(* CODESYS project SGS V4.project
   Description: Diese Software wurde während der Bachelorarbeit für das Strom-Generatorsystem entwickelt.
   Company: Zoyce GmbH
   Version: 4.0
   Title: Strom-Generatorsystem
   Author: Julian Städeli

Project tree, tasks and I/O mapping:
  PLC_AC500_V3 : PM5052-R-ETH, ABB AG, order no. 1SAP124100R0x72, version 3.7.0.0
    application Application
      libraries: Util, * (System); CAA Mathematics, * (CAA Technical Workgroup); VisuElemBase, 4.4.0.0 (System); OnboardIO, * (ABB); VisuDialogs, * (System); SysFile, * (System); SysTimeRtc, * (System); CAA File, * (CAA Technical Workgroup); CAA DTUtil Extern, * (CAA Technical Workgroup); CAA Types Extern, * (CAA Technical Workgroup); SysTime, 3.5.17.0 (System); CAA Memory, * (CAA Technical Workgroup); SysTypes Interfaces, * (System); MQTT Client SL, 1.9.0.0 (CODESYS)
      task Task (cyclic, interval 10 ms, priority 14, watchdog t#20ms x 1) calls Ueberwachung, SunSpec_client, Inverter, Berechnungen, Systemzustand, MQTTDataLogger
      task VISU_TASK (cyclic, interval 100 ms, priority 16) calls VisuElems.Visu_Prg
      CheckConfigurationObject
      program PLC_PRG [ST]
      Diagnosis/
        text list Diag_IO_Bus
        text list Diag_V3_PLC
      trace Trace_Drehzahl (task Task): GV.sys_Drehzahl, GV.sys_Drehzahl_Sensor, GV.sys_Drehzahl_Estimator, GV.sys_Drehzahl_Rechner
      trace Trace_Leistung (task Task): GV.r_LeistungAC, GV.r_LeistungDC
      Symbols
    OnBoard_IO : 12DI/6DO-R/2DC, ABB AG, version 3.7.0.0
        unmapped channels: Fast inputs DI0-DI3, %IB1 Fast inputs DI4-DI7, Standard inputs DI8-DI11, Digital configurable inputs DC12-DC13, Relay outputs NO0-NO3, Relay outputs NO4-NO5 - Digital configurable outputs DC12-DC13
    IO_Bus : I/O-Bus, ABB AG, version 3.7.0.0
    Interfaces : Schnittstellen, ABB AG, version 3.7.0.0
      OptionSlot_1
      OptionSlot_2
      OptionSlot_3
      Ethernet : Ethernet, ABB AG, version 3.7.0.0
        ETH1 : IP-Einstellungen, ABB AG, version 3.7.0.0
          NetConfig : NetzKonfig, ABB AG, version 3.7.0.0
          Web_Server : Webserver, ABB AG, version 3.7.0.0
        Protocols : Client-Protokolle, ABB AG, version 3.7.0.0
          Modbus_TCP_IP_Client : Modbus TCP/IP Client, ABB AG, version 3.7.0.0
    OnBoard_RTC : OnBoardRTC, ABB AG, version 3.7.0.0
  libraries: VisuSymbols, 4.4.0.0 (System); VisuDialogs, * (System); CmpBitmapPool, 3.5.17.0 (System); SysFile, 3.5.17.0 (System); SysFile, 1.0.3.1 (ABB); CAA DTUtil Extern, 3.5.17.0 (CAA Technical Workgroup); SysTypes, 3.1.2.0 (System); SysTypes Interfaces, * (System); SysTimeRtc, 3.5.17.0 (System); CAA File, 3.5.19.0 (CAA Technical Workgroup); MQTT Client SL, 1.9.0.0 (CODESYS)
  global variables GV
  program Schaltlogik [FBD]
  program Ueberwachung [FBD]
  text list GlobalTextList
  program SunSpec_client [FBD]
  data type SunSpec_Model_Inverter1
  SunSpec_Translator/
    function block SunSpec_Write [FBD]
    function block SunSpec_Model_Inverter [ST]
    function block SunSpec_Model_Settings [ST]
    function block SunSpec_Model_Status [ST]
    function block SunSpec_Model_Controls [ST]
    function block SunSpec_Model_MPPT [ST]
    function block SunSpec_Model_Meter [ST]
  program Inverter [ST]
  program Berechnungen [ST]
  image pool ImagePool
  Visualisierung/
    visualisation Uebersicht
    visualisation Elektrotechnik
    visualisation System
    visualisation Parameter
    visualisation Show
    visualisation Logging
    visualisation Info
  5ce3da45-db07-42e7-a21c-a00fff4ed8f6|C:\Users\julia\OneDrive - FHNW\Pro5E\Bilder\Uebersicht Visu.png
  program Systemzustand [ST]
  function block FB_DataLogger [ST]
  5ce3da45-db07-42e7-a21c-a00fff4ed8f6|C:\Users\julia\Downloads\Visu_Show.png
  function WSTRING_TO_BYTEARRAY_UTF8 [ST]
  function block FB_MQTT_Logger [ST]
  function WSTRING_Concat [ST]
  program MQTTDataLogger [ST]
*)

// SunSpec_Model_Inverter1
TYPE SunSpec_Model_Inverter1 :
STRUCT
	ID	:INT;
	Length	:INT;
	AC_Current	:INT;
	Phase_A_Current	:REAL;
	Phase_B_Current	:REAL;
	Phase_C_Current	:REAL;
	
	Phase_Voltage_AB	:REAL;
	Phase_Voltage_BC	:REAL;
	Phase_Voltage_CA	:REAL;
	Phase_Voltage_AN	:REAL;
	Phase_Voltage_BN	:REAL;
	Phase_Voltage_CN	:REAL;
	
	AC_Power	:REAL;
	AC_Frequency	:REAL;
	
	AC_Apparent_Power	:REAL;
	AC_Reactive_Power	:REAL;
	AC_PowerFactor		:REAL;
	AC_Energy			:REAL;
	
	DC_Power	:REAL;
	Temperature :REAL;

	
	
	
	
	
	
	
	
	
	
	
	
END_STRUCT
END_TYPE

// GV
{attribute 'qualified_only'}
(*
Diese Software rurde für die Bachelorarbeit "Stromerzeugungssystem für ein Kleinwasserkraftwerk" 
an der Fachhochschule Nordwestschweiz (FHNW) entwickelt.

Diplomand:		Julian Städeli
				julian.staedeli@students.fhnw.ch	|	julian@staedelis.com
Dozent:			Georg Traxler-Samek
				georg.traxlersamek@fhnw.ch
				
*)

VAR_GLOBAL
	
// Inputs
I_Notaus 			AT %IX0.0		:BOOL;		// I0 Not-Aus Kontakt
I_Steuerspannung 	AT %IX0.1		:BOOL;		// I1 Ausgang Relais Steuerspannung
I_Einschalten 		AT %IX0.2		:BOOL;		// I2 Kontakt Einschalttaster
I_Ausschalten 		AT %IX0.3		:BOOL;		// I3 Kontakt Ausschalttaster
I_Sensor_Drehzahl 	AT %IX1.0		:BOOL;		// I4 Kontakt Sensor, Induktiver Näherungsschalter
I_Hauptschuetz 		AT %IX1.1		:BOOL;		// I5 Hilfskontakt Hauptschütz
I_Ladeschuetz 		AT %IX1.2		:BOOL;		// I6 Hilfskontakt Ladeschütz
I_Motorschutz 		AT %IX1.3		:BOOL;		// I7 Hilfskontakt Motorschutzschalter
I_Temperatur 		AT %IX2.0		:BOOL;		// I8 Thermokontakt im Generator

I_Counter							:UDINT;		// Fast Counter für Sensor

 //AT %IX3.0

// Outputs
O_Steuerspannung	AT %QX0.1		:BOOL;		// NO1 Relais Steuerspannung
O_Infolampe			AT %QX0.2		:BOOL;		// NO2 Infolampe auf Bedienfeld 
O_Hauptschuetz 		AT %QX0.3		:BOOL;		// NO3 Hauptschütz
O_Ladeschuetz		AT %QX1.0		:BOOL;		// NO4 Ladeschütz


// Störungen
stoerung_Notaus				:BOOL;
stoerung_Steuerspannung		:BOOL;
stoerung_Hauptschuetz		:BOOL;
stoerung_Ladeschuetz		:BOOL;
stoerung_Motorschutz		:BOOL;
stoerung_Inverter			:BOOL;
stoerung_Temperatur			:BOOL;

stoerung_Drehzahl			:BOOL;
sammelstoerung				:BOOL;
stoerung_quittieren			:BOOL;

stoerung_Modbus_Lesen		:BOOL;
stoerung_Modbus_Schreiben	:BOOL;
stoerung_MQTT				:BOOL;


// Zustände System
sys_Einschalten				:BOOL;				// Einschaltbefehl
sys_Ausschalten				:BOOL;				// Auschaltbefehl

sys_aus						:BOOL :=TRUE;		// System ist aus: Inverter Heruntergefahren, Schütze offen, Geni im Leerlauf
sys_start					:BOOL;				// Einschaltprozess mit Ladeschaltung und Hochfahren des Inverters
sys_bereit					:BOOL;				// System bereit zum Produzieren
sys_betrieb					:BOOL;				// System läuft 
sys_herunterfahren			:BOOL;				// System wird heruntergefahren

sys_MPPT_aktiv				:BOOL;		// System soll über MPPT arbeiten / befindet sich im Automatikbetrieb
sys_MPP_erreicht			:BOOL;				// Gibt an, ob sich der Tracker am MPP befindet.
sys_LeistungBegrenzung 		:UINT;				// Die eingestellte Leistung, die dem Inverter als Begrenzung übergeben wird (Wert 100 = 10% von 3000W)
			
sys_Drehzahl_Sensor			:REAL;				// Berechnete Drehzahl über Sensor
sys_Drehzahl_Estimator		:REAL;				// Berechnete Drehzahl über der gemessenen Spannung
sys_Drehzahl_Rechner		:REAL;				// Berechnete Drehzahl über Ersatzschaltbild
sys_Drehzahl				:REAL; 				// Systemdrehzahl, die von dem Programm genutzt wird (über Parameter einstellbar)
sys_Drehzahl_Wasserrad		:REAL;				// Berechnete Drehzahl des Wasserrads

// Inverter

// Zustände Inverter
r_StateCode					:STRING; 			// Aus / Standby / Startet / Arbeitet
r_Status					:STRING;
r_Begrenzung				:STRING; 			// Ein / Aus

inv_herunterfahren			:BOOL;				// Inverter soll ausgeschaltet werden
inv_ein						:BOOL;				// Ist eingeschaltet
inv_bereit					:BOOL;				// Ist hochgefahren 
inv_betrieb					:BOOL;				// produziert
inv_leerlauf				:BOOL;				// Ist eingekoppelt aber keine produktion
inv_standby					:BOOL;
inv_fehler					:BOOL;
inv_MaxLeistungEingestellt 	:REAL;				// Eingestellte Leistungsbegrenzung



// Visu
v_LeistungBegrenzung		:UINT;				// Eingestellte Leistung über Visu [W]
v_LeistungBegrenzung_ein	:BOOL;				// Begrenzung mit Visu forcieren

v_Einschalten				:BOOL;				// Einschaltbefehl über Visu
v_Ausschalten				:BOOL;				// Ausschaltbefehl über Visu
v_Notaus					:BOOL;				// Notaus üner Visu
v_Geni_lauft				:BOOL;				// Es wird eine Drehzahl gemessen


	// Modbus 
inv_IP						:STRING;			// IP-Adresse des Inverter, z. B. '192.168.0.51'


	// Daten Modbus (readings)
	//Inverter
r_StromPhaseA				:REAL;		// [A]
r_StromPhaseB				:REAL;		// [A]
r_StromPhaseC				:REAL;		// [A]
r_StrangspannungA			:REAL;		// [V]
r_StrangspannungB			:REAL;		// [V]
r_StrangspannungC			:REAL;		// [V]
r_SpannungPCC				:REAL;		// [V]

r_Frequenz					:REAL;		// [Hz]
r_LeistungAC				:REAL;		// [W]
r_PF						:REAL;
r_Energie					:REAL;		// [Wh]

r_StromDC					:REAL;		// [A]
r_SpannungDC				:REAL;		// [V]
r_LeistungDC				:REAL;		// [W]
r_EnergieDC					:REAL;		// [Wh]		

r_Temperatur				:REAL;		// [°C]

r_MaxLeistung				:REAL;		// [W]

 // Smartmeter
 r_sm_Leistung				:REAL;


	// Befehle Modbus (write)
w_Einschalten				:UINT :=1;	// Inverter soll Einschalten
w_LeistungBegrenzung		:UINT;		// Entweder über Visu oder MPPT vorgegebene Leistungsbegrenzung [%]
w_RampTime	 				:UINT;		// Zeitintervall von einem punkt zum nächsten (funktioniert nicht) [s]
w_Standby					:UINT;		// Inverter soll Ausschalten

	// Überprüfung der Eingestellten Werte
r_Einschalten				:INT;
r_LeistungBegrenzung		:REAL;		
r_RampTime					:REAL;	
r_Standby					:STRING;	




// Parameter
p_Inverter_IP		:STRING :='192.168.178.45';		// IP-Adresse des Inverter, z. B. '192.168.0.51'

p_Drehzahl_soll		:INT :=360;						// Sollwert für Drehzahlregulierung [rpm]					
p_Drehzahl_Toleranz	:INT :=5;						// Angenommene Ungenauigkeit [rpm]
p_Drehzahl_max		:INT :=690;						// Maximal erlaubte Drehzahl [rpm]
p_Drehzahl_min		:INT :=200;						// Minimal benötigte Drehzahl [rpm]
p_Sensor_Impulse	:INT := 4;						// Anzahl Impulse pro rpm die der Sensor liefert [1/rpm]
p_Sensor_Intervall	:TIME := T#1S;					// Wie lange die Impulse vor der Berechnung gemacht werden

p_Leistung_Init		:UINT := 200;					// Mit welcher Leistung gestartet wird [100.00% = 10000]
p_Leistung_Toleranz	:REAL :=30;						// Erlaubte Abweichung, damit es als erreicht gilt [W]
p_Leistung_Anpassung :REAL := 10;					// Leistungsanpassungsschritt [00.10%= 10]

p_MPPT_Intervall	:TIME := T#3S;					// Wie lange gewartet wird, bis MPP einen nächsten Schritt macht [s]
p_MPPT_Timeout		:TIME :=T#3S;					// Wie lange, bis die Leistung als  nicht erreicht betrachtet wird [s]

p_Automatik			:BOOL := TRUE; 					// System fährt selbständig hoch und runter

p_Herunterfahren_Intervall	:TIME := T#1S;			// Wie langae zwischen den Schritten gewartet wird [s]

timenow			:DATE_AND_TIME;


// Show
v_speicher_start	:BOOL := TRUE;
v_Kaffeemaschine :REAL;
v_speicher :REAL :=0;

log_time :ARRAY[1..2000] OF REAL;
log_DrehzahlSoll :ARRAY[1..2000] OF REAL;
log_DrehzahlIst :ARRAY[1..2000] OF REAL;
log_Leistung :ARRAY[1..2000] OF REAL;

END_VAR

// Ueberwachung
PROGRAM Ueberwachung
VAR
	zeit_bis_stoerung :TIME :=t#1s;
	RS_Notaus: RS;
	TON_stoerung_Steuerspannung: TON;
	RS_stoerung_Steuerspannung: SR;
	TON_stoerung_Hauptschuetz: TON;
	RS_stoerung_Hauptschuetz: RS;
	TON_stoerung_Ladeschuetz: TON;
	RS_stoerung_Ladeschuetz: RS;
	RS_Motorschutz: RS;
	RS_Sammelstoerung: RS;
	TON_quittieren: TON;
	RS_Drehzahl: RS;
	TON_Drehzahl: TON;
	RS_Temperatur: RS;
	SR_Notaus: SR;
	SR_stoerung_Steuerspannung: SR;
	SR_stoerung_Hauptschuetz: SR;
	SR_stoerung_Ladeschuetz: SR;
	SR_Motorschutz: SR;
	SR_Temperatur: SR;
	SR_Drehzahl: SR;
	SR_Sammelstoerung: SR;
END_VAR

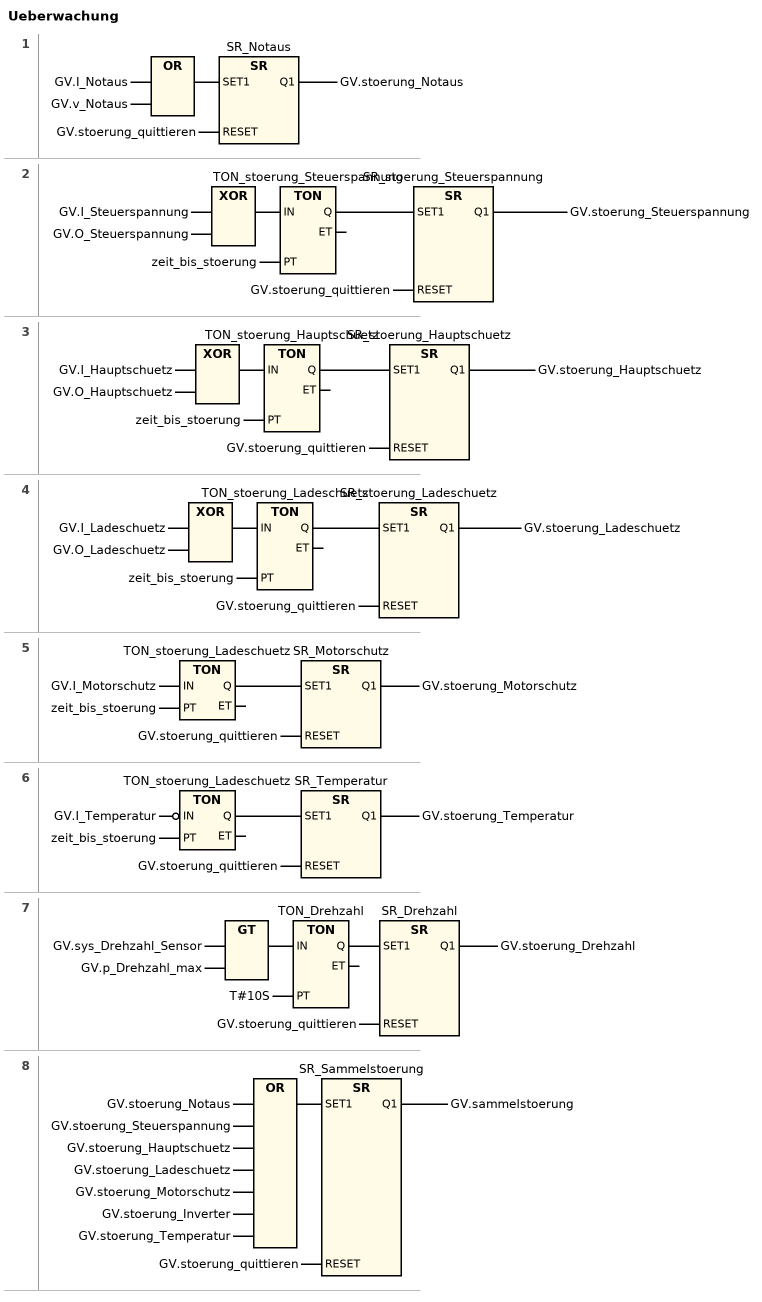
// NETWORK 1
SR_Notaus(SET1 := GV.I_Notaus OR GV.v_Notaus, RESET := GV.stoerung_quittieren); // SR
GV.stoerung_Notaus := SR_Notaus.Q1;

// NETWORK 2
TON_stoerung_Steuerspannung(IN := GV.I_Steuerspannung XOR GV.O_Steuerspannung, PT := zeit_bis_stoerung); // TON
SR_stoerung_Steuerspannung(SET1 := TON_stoerung_Steuerspannung.Q, RESET := GV.stoerung_quittieren); // SR
GV.stoerung_Steuerspannung := SR_stoerung_Steuerspannung.Q1;

// NETWORK 3
TON_stoerung_Hauptschuetz(IN := GV.I_Hauptschuetz XOR GV.O_Hauptschuetz, PT := zeit_bis_stoerung); // TON
SR_stoerung_Hauptschuetz(SET1 := TON_stoerung_Hauptschuetz.Q, RESET := GV.stoerung_quittieren); // SR
GV.stoerung_Hauptschuetz := SR_stoerung_Hauptschuetz.Q1;

// NETWORK 4
TON_stoerung_Ladeschuetz(IN := GV.I_Ladeschuetz XOR GV.O_Ladeschuetz, PT := zeit_bis_stoerung); // TON
SR_stoerung_Ladeschuetz(SET1 := TON_stoerung_Ladeschuetz.Q, RESET := GV.stoerung_quittieren); // SR
GV.stoerung_Ladeschuetz := SR_stoerung_Ladeschuetz.Q1;

// NETWORK 5
TON_stoerung_Ladeschuetz(IN := GV.I_Motorschutz, PT := zeit_bis_stoerung); // TON
SR_Motorschutz(SET1 := TON_stoerung_Ladeschuetz.Q, RESET := GV.stoerung_quittieren); // SR
GV.stoerung_Motorschutz := SR_Motorschutz.Q1;

// NETWORK 6
TON_stoerung_Ladeschuetz(IN := NOT GV.I_Temperatur, PT := zeit_bis_stoerung); // TON
SR_Temperatur(SET1 := TON_stoerung_Ladeschuetz.Q, RESET := GV.stoerung_quittieren); // SR
GV.stoerung_Temperatur := SR_Temperatur.Q1;

// NETWORK 7
TON_Drehzahl(IN := GV.sys_Drehzahl_Sensor > GV.p_Drehzahl_max, PT := T#10S); // TON
SR_Drehzahl(SET1 := TON_Drehzahl.Q, RESET := GV.stoerung_quittieren); // SR
GV.stoerung_Drehzahl := SR_Drehzahl.Q1;

// NETWORK 8
SR_Sammelstoerung(SET1 := GV.stoerung_Notaus OR GV.stoerung_Steuerspannung OR GV.stoerung_Hauptschuetz OR GV.stoerung_Ladeschuetz OR GV.stoerung_Motorschutz OR GV.stoerung_Inverter OR GV.stoerung_Temperatur, RESET := GV.stoerung_quittieren); // SR
GV.sammelstoerung := SR_Sammelstoerung.Q1;

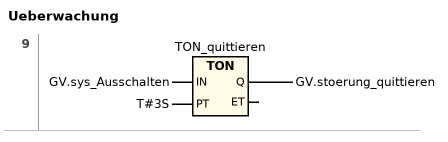
// NETWORK 9
TON_quittieren(IN := GV.sys_Ausschalten, PT := T#3S); // TON
GV.stoerung_quittieren := TON_quittieren.Q;

END_PROGRAM

// SunSpec_client
PROGRAM SunSpec_client
VAR
	inverterIP :STRING := GV.p_Inverter_IP;
// SunSpec Adressen für das Auslesen
	// SunSpec_Adr_Model_Common :WORD := 40003;
	SunSpec_Adr_Model_Inverter :WORD := 40070;
	// SunSpec_Adr_Model_Nameplate :WORD := 40122;
	SunSpec_Adr_Model_Settings :WORD := 40150;
	SunSpec_Adr_Model_Status	:WORD := 40182;
	SunSpec_Adr_Model_Controls :WORD := 40228;
	SunSpec_Adr_Model_MPPT		:WORD := 40254;
	SunSpec_Adr_Model_AC_Meter	:WORD := 40070;
// Buffer für Lesedaten
	inverterData_Inverter AT %MW10 : ARRAY[1..50] OF INT;
	inverterData_Settings AT %MW60 :ARRAY [1..30] OF INT;
	inverterData_Status AT %MW90 :ARRAY [1..50] OF INT;
	inverterData_Controls AT %MW140:ARRAY [1..30] OF INT;
	inverterData_MPPT AT %MW170 :ARRAY [1..30] OF INT;	
	meterData_Main AT %MW200 :ARRAY [1..75] OF INT;

	
// SunSpec Adressen für das Schreiben	
	SunSpec_Adr_Connection	:WORD := 40232;
	SunSpec_Adr_MaxPower	:WORD := 40233;
	SunSpec_Adr_RampTime		:WORD := 40236;
	SunSpec_Adr_Throttle	:WORD := 40237;
// Buffer für Schreibdaten
	inverterCommand_Connection 	AT %MW1		:UINT := GV.w_Einschalten;
	inverterCommand_maxPower 	AT %MW2		:UINT := GV.w_LeistungBegrenzung;
	inverterCommand_RampTime 	AT %MW3		:UINT := GV.w_RampTime;
	inverterCommand_Throttle 	AT %MW4		:UINT :=1;

	clk_Pulse :TIME := T#900MS;
	
	clock: BLINK;
	SunSpec_Inverter: modTcpMast2;
	SunSpec_Settings: ModTcpMast2;
	SunSpec_Controls: modTcpMast2;
	SunSpec_MPPT: modTcpMast2;
	SunSpec_Status: modTcpMast2;
	SunSpec_Write: modTcpMast2;
	SunSpec_Model_Inverter_0: SunSpec_Model_Inverter;
	SunSpec_Model_Settings_0: SunSpec_Model_Settings;
	SunSpec_Model_Status_0: SunSpec_Model_Status;
	SunSpec_Model_Controls_0: SunSpec_Model_Controls;
	SunSpec_Model_MPPT_0: SunSpec_Model_MPPT;
	R_TRIG_0: R_TRIG;
	SunSpec_Write1: modTcpMast2;
	SunSpec_Write2: modTcpMast2;
	SunSpec_Write_0: SunSpec_Write;
	SunSpec_Meter_main: modTcpMast2;
	SunSpec_Meter_Generator: modTcpMast2;
	SunSpec_Model_Meter_main: SunSpec_Model_Meter;
	SunSpec_Model_Meter_generator: SunSpec_Model_Meter;
END_VAR

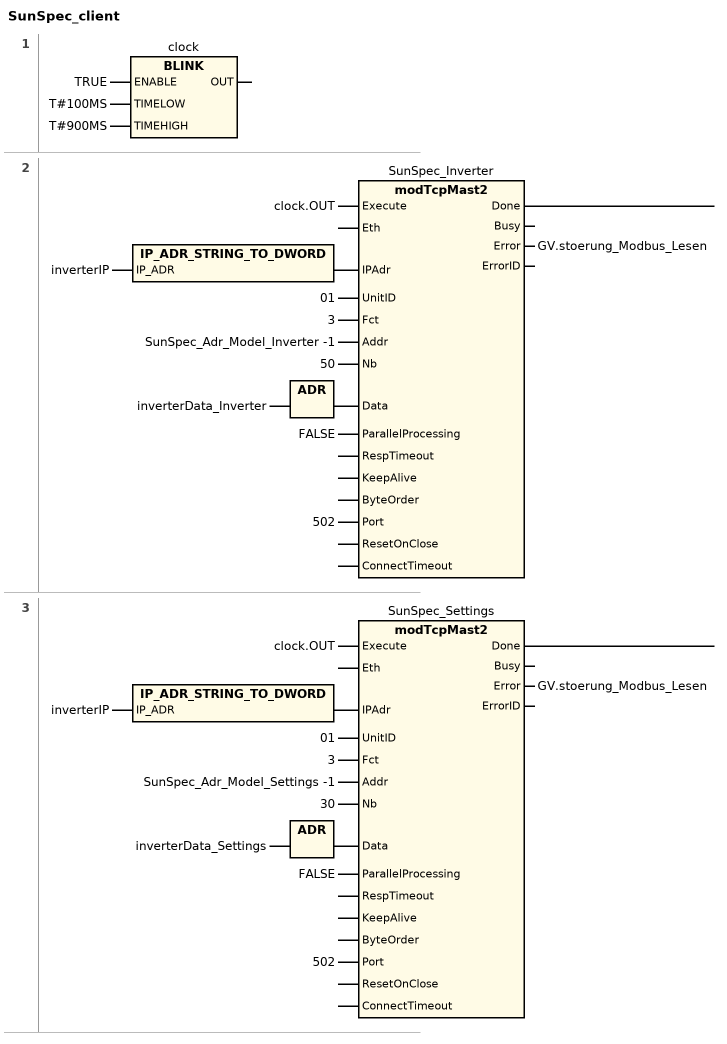
// NETWORK 1
clock(ENABLE := TRUE, TIMELOW := T#100MS, TIMEHIGH := T#900MS); // BLINK

// NETWORK 2
SunSpec_Inverter(
    Execute := clock.OUT,
    IPAdr := IP_ADR_STRING_TO_DWORD(IP_ADR := inverterIP),
    UnitID := 01,
    Fct := 3,
    Addr := SunSpec_Adr_Model_Inverter -1,
    Nb := 50,
    Data := ADR(inverterData_Inverter),
    ParallelProcessing := FALSE,
    Port := 502,
    Error => GV.stoerung_Modbus_Lesen); // modTcpMast2

// NETWORK 3
SunSpec_Settings(
    Execute := clock.OUT,
    IPAdr := IP_ADR_STRING_TO_DWORD(IP_ADR := inverterIP),
    UnitID := 01,
    Fct := 3,
    Addr := SunSpec_Adr_Model_Settings -1,
    Nb := 30,
    Data := ADR(inverterData_Settings),
    ParallelProcessing := FALSE,
    Port := 502,
    Error => GV.stoerung_Modbus_Lesen); // modTcpMast2

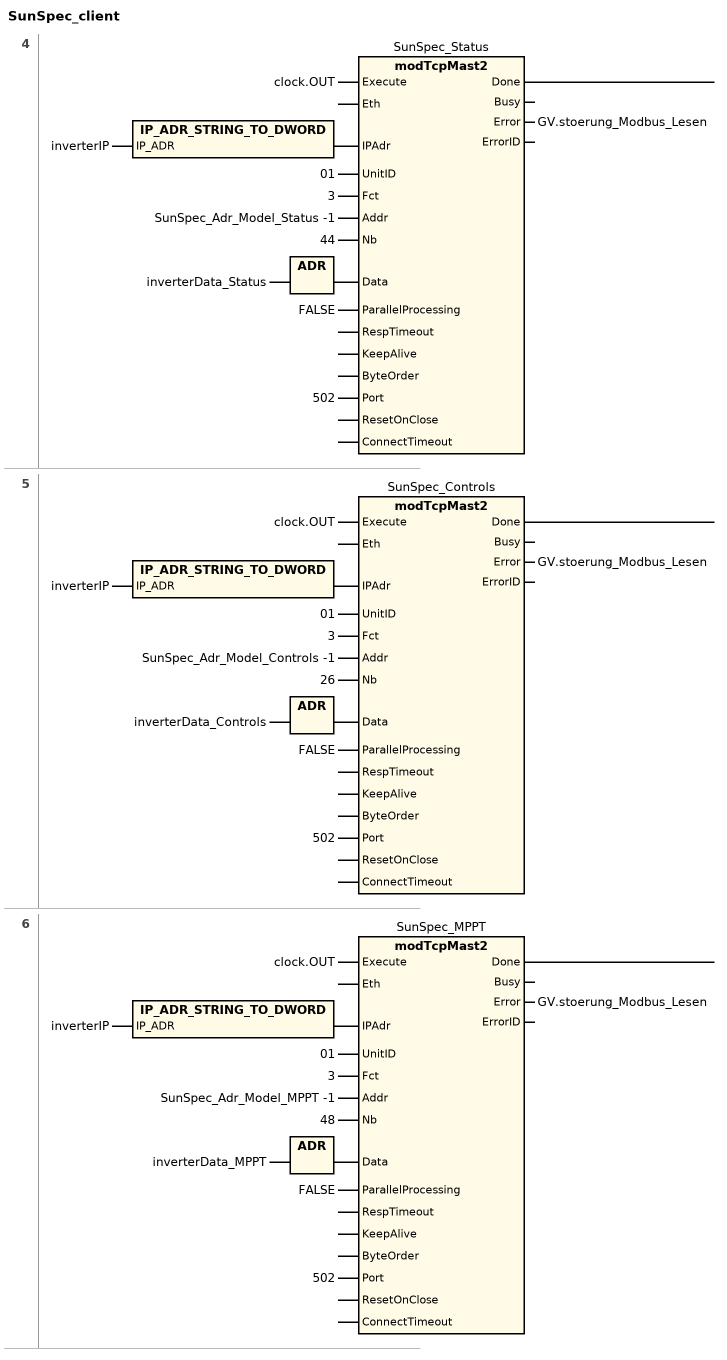
// NETWORK 4
SunSpec_Status(
    Execute := clock.OUT,
    IPAdr := IP_ADR_STRING_TO_DWORD(IP_ADR := inverterIP),
    UnitID := 01,
    Fct := 3,
    Addr := SunSpec_Adr_Model_Status -1,
    Nb := 44,
    Data := ADR(inverterData_Status),
    ParallelProcessing := FALSE,
    Port := 502,
    Error => GV.stoerung_Modbus_Lesen); // modTcpMast2

// NETWORK 5
SunSpec_Controls(
    Execute := clock.OUT,
    IPAdr := IP_ADR_STRING_TO_DWORD(IP_ADR := inverterIP),
    UnitID := 01,
    Fct := 3,
    Addr := SunSpec_Adr_Model_Controls -1,
    Nb := 26,
    Data := ADR(inverterData_Controls),
    ParallelProcessing := FALSE,
    Port := 502,
    Error => GV.stoerung_Modbus_Lesen); // modTcpMast2

// NETWORK 6
SunSpec_MPPT(
    Execute := clock.OUT,
    IPAdr := IP_ADR_STRING_TO_DWORD(IP_ADR := inverterIP),
    UnitID := 01,
    Fct := 3,
    Addr := SunSpec_Adr_Model_MPPT -1,
    Nb := 48,
    Data := ADR(inverterData_MPPT),
    ParallelProcessing := FALSE,
    Port := 502,
    Error => GV.stoerung_Modbus_Lesen); // modTcpMast2

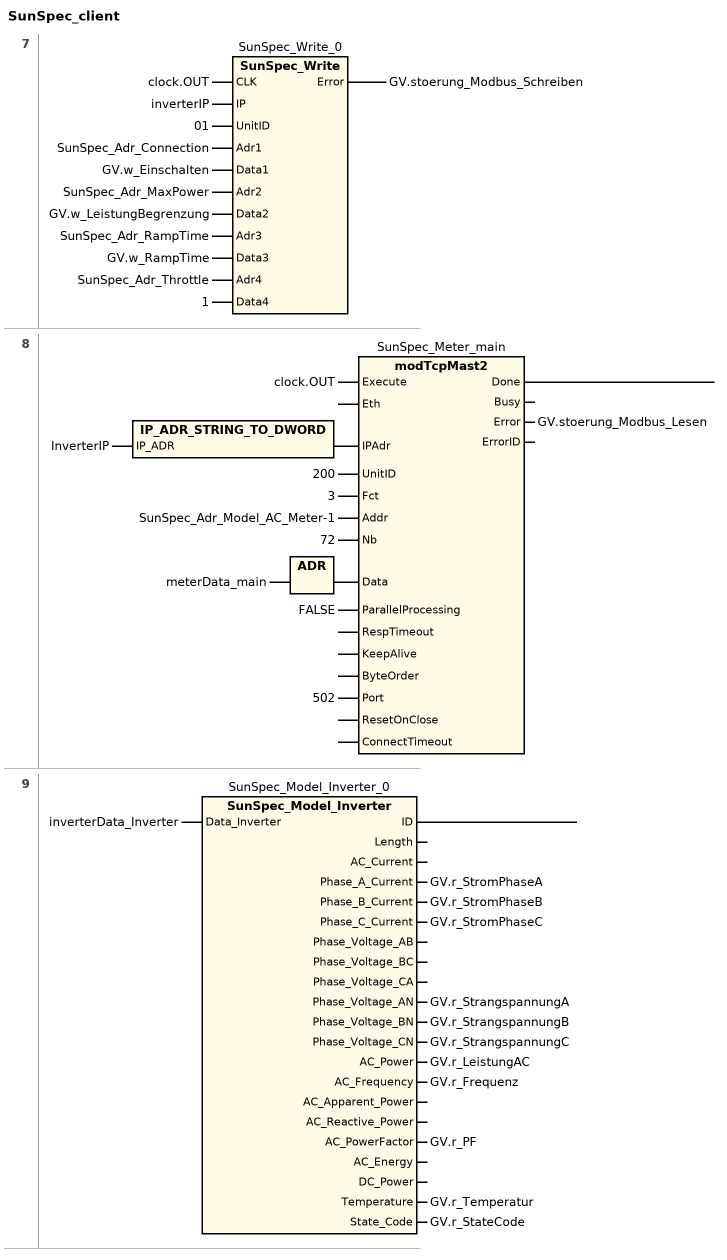
// NETWORK 7
SunSpec_Write_0(
    CLK := clock.OUT,
    IP := inverterIP,
    UnitID := 01,
    Adr1 := SunSpec_Adr_Connection,
    Data1 := GV.w_Einschalten,
    Adr2 := SunSpec_Adr_MaxPower,
    Data2 := GV.w_LeistungBegrenzung,
    Adr3 := SunSpec_Adr_RampTime,
    Data3 := GV.w_RampTime,
    Adr4 := SunSpec_Adr_Throttle,
    Data4 := 1); // SunSpec_Write
GV.stoerung_Modbus_Schreiben := SunSpec_Write_0.Error;

// NETWORK 8
SunSpec_Meter_main(
    Execute := clock.OUT,
    IPAdr := IP_ADR_STRING_TO_DWORD(IP_ADR := InverterIP),
    UnitID := 200,
    Fct := 3,
    Addr := SunSpec_Adr_Model_AC_Meter-1,
    Nb := 72,
    Data := ADR(meterData_main),
    ParallelProcessing := FALSE,
    Port := 502,
    Error => GV.stoerung_Modbus_Lesen); // modTcpMast2

// NETWORK 9
SunSpec_Model_Inverter_0(
    Data_Inverter := inverterData_Inverter,
    Phase_A_Current => GV.r_StromPhaseA,
    Phase_B_Current => GV.r_StromPhaseB,
    Phase_C_Current => GV.r_StromPhaseC,
    Phase_Voltage_AN => GV.r_StrangspannungA,
    Phase_Voltage_BN => GV.r_StrangspannungB,
    Phase_Voltage_CN => GV.r_StrangspannungC,
    AC_Power => GV.r_LeistungAC,
    AC_Frequency => GV.r_Frequenz,
    AC_PowerFactor => GV.r_PF,
    Temperature => GV.r_Temperatur,
    State_Code => GV.r_StateCode); // SunSpec_Model_Inverter

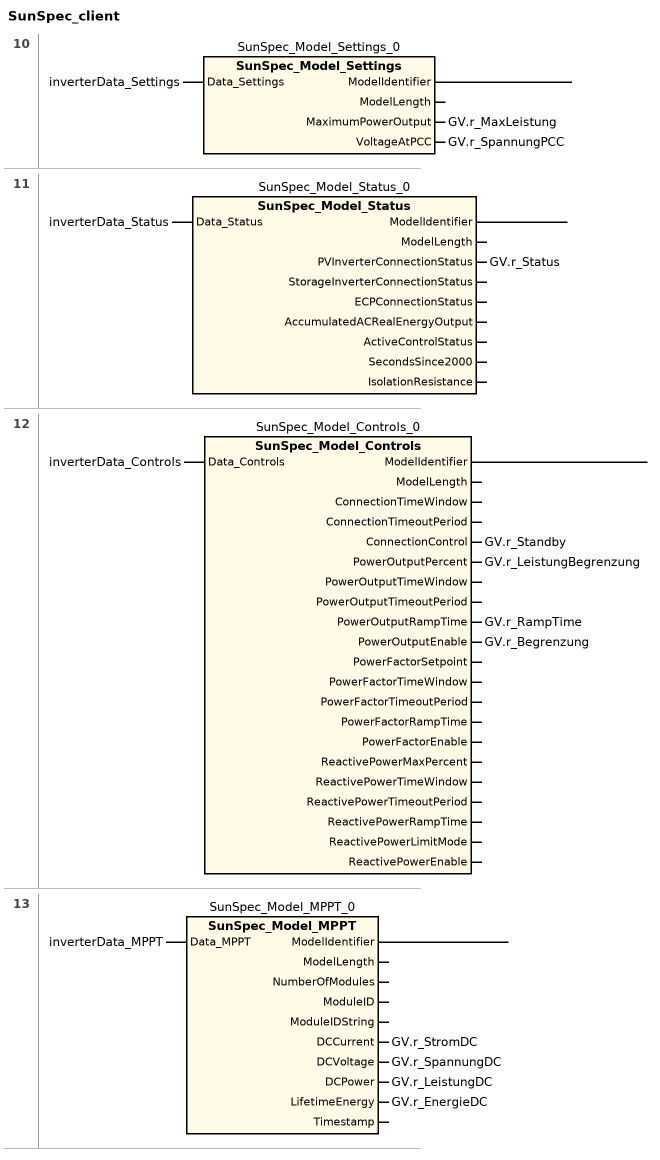
// NETWORK 10
SunSpec_Model_Settings_0(
    Data_Settings := inverterData_Settings,
    MaximumPowerOutput => GV.r_MaxLeistung,
    VoltageAtPCC => GV.r_SpannungPCC); // SunSpec_Model_Settings

// NETWORK 11
SunSpec_Model_Status_0(Data_Status := inverterData_Status, PVInverterConnectionStatus => GV.r_Status); // SunSpec_Model_Status

// NETWORK 12
SunSpec_Model_Controls_0(
    Data_Controls := inverterData_Controls,
    ConnectionControl => GV.r_Standby,
    PowerOutputPercent => GV.r_LeistungBegrenzung,
    PowerOutputRampTime => GV.r_RampTime,
    PowerOutputEnable => GV.r_Begrenzung); // SunSpec_Model_Controls

// NETWORK 13
SunSpec_Model_MPPT_0(
    Data_MPPT := inverterData_MPPT,
    DCCurrent => GV.r_StromDC,
    DCVoltage => GV.r_SpannungDC,
    DCPower => GV.r_LeistungDC,
    LifetimeEnergy => GV.r_EnergieDC); // SunSpec_Model_MPPT

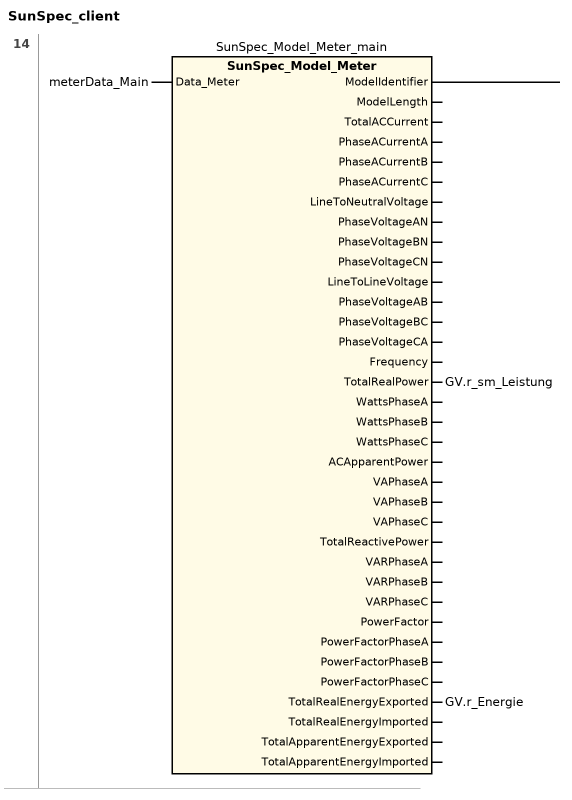
// NETWORK 14
SunSpec_Model_Meter_main(
    Data_Meter := meterData_Main,
    TotalRealPower => GV.r_sm_Leistung,
    TotalRealEnergyExported => GV.r_Energie); // SunSpec_Model_Meter

END_PROGRAM

// SunSpec_Translator/SunSpec_Write
FUNCTION_BLOCK SunSpec_Write
VAR_INPUT
	CLK		:BOOL;
	IP		:STRING;
	UnitID	:BYTE;
	
	Adr1	:WORD;
	Data1	:INT;
	Adr2	:WORD;
	Data2	:INT;
	Adr3	:WORD;
	Data3	:INT;
	Adr4	:WORD;
	Data4	:INT;
// 	Adr5	:WORD;
// 	Data5	:INT;
	
END_VAR
VAR_OUTPUT
	Error	:BOOL;
END_VAR
VAR
	modTcpMast2_0: modTcpMast2;
	modTcpMast2_1: modTcpMast2;
	modTcpMast2_2: modTcpMast2;
	modTcpMast2_3: modTcpMast2;
	modTcpMast2_4: modTcpMast2;
END_VAR

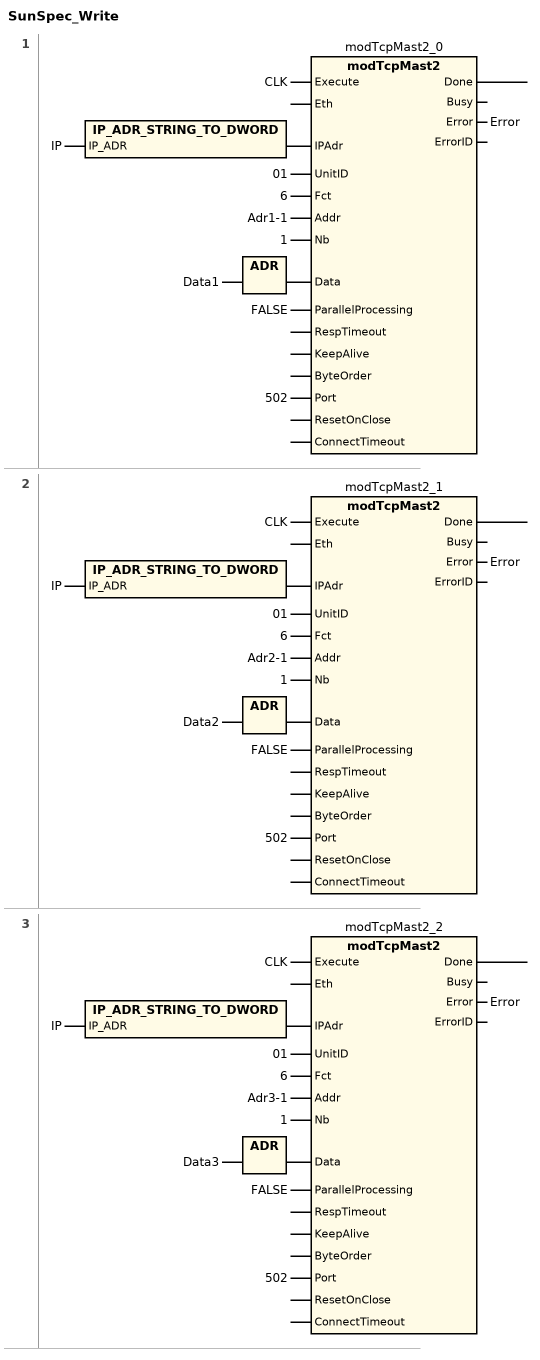
// NETWORK 1
modTcpMast2_0(
    Execute := CLK,
    IPAdr := IP_ADR_STRING_TO_DWORD(IP_ADR := IP),
    UnitID := 01,
    Fct := 6,
    Addr := Adr1-1,
    Nb := 1,
    Data := ADR(Data1),
    ParallelProcessing := FALSE,
    Port := 502,
    Error => Error); // modTcpMast2

// NETWORK 2
modTcpMast2_1(
    Execute := CLK,
    IPAdr := IP_ADR_STRING_TO_DWORD(IP_ADR := IP),
    UnitID := 01,
    Fct := 6,
    Addr := Adr2-1,
    Nb := 1,
    Data := ADR(Data2),
    ParallelProcessing := FALSE,
    Port := 502,
    Error => Error); // modTcpMast2

// NETWORK 3
modTcpMast2_2(
    Execute := CLK,
    IPAdr := IP_ADR_STRING_TO_DWORD(IP_ADR := IP),
    UnitID := 01,
    Fct := 6,
    Addr := Adr3-1,
    Nb := 1,
    Data := ADR(Data3),
    ParallelProcessing := FALSE,
    Port := 502,
    Error => Error); // modTcpMast2

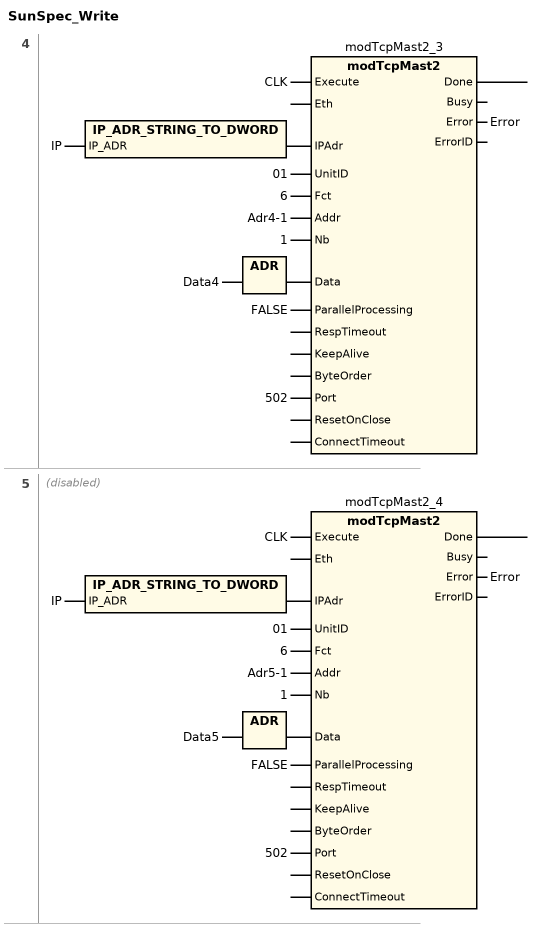
// NETWORK 4
modTcpMast2_3(
    Execute := CLK,
    IPAdr := IP_ADR_STRING_TO_DWORD(IP_ADR := IP),
    UnitID := 01,
    Fct := 6,
    Addr := Adr4-1,
    Nb := 1,
    Data := ADR(Data4),
    ParallelProcessing := FALSE,
    Port := 502,
    Error => Error); // modTcpMast2

// NETWORK 5 (disabled)
// modTcpMast2_4(
//     Execute := CLK,
//     IPAdr := IP_ADR_STRING_TO_DWORD(IP_ADR := IP),
//     UnitID := 01,
//     Fct := 6,
//     Addr := Adr5-1,
//     Nb := 1,
//     Data := ADR(Data5),
//     ParallelProcessing := FALSE,
//     Port := 502,
//     Error => Error); // modTcpMast2

END_FUNCTION_BLOCK

// SunSpec_Translator/SunSpec_Model_Inverter
FUNCTION_BLOCK SunSpec_Model_Inverter
VAR_INPUT
	Data_Inverter :ARRAY [1..50] OF INT;
END_VAR
VAR_OUTPUT
	ID	:INT;
	Length	:INT;
	AC_Current	:REAL;
	Phase_A_Current	:REAL;
	Phase_B_Current	:REAL;
	Phase_C_Current	:REAL;
	
	Phase_Voltage_AB	:REAL;
	Phase_Voltage_BC	:REAL;
	Phase_Voltage_CA	:REAL;
	Phase_Voltage_AN	:REAL;
	Phase_Voltage_BN	:REAL;
	Phase_Voltage_CN	:REAL;
	
	AC_Power	:REAL;
	AC_Frequency	:REAL;
	
	AC_Apparent_Power	:REAL;
	AC_Reactive_Power	:REAL;
	AC_PowerFactor		:REAL;
	AC_Energy			:REAL;
	
	DC_Power	:REAL;
	Temperature :REAL;
	
	State_Code	:STRING;

	

END_VAR


VAR
	Status		:INT;
	sf_AC_Current :REAL;
	sf_AC_Voltage :REAL;
	sf_AC_Power :REAL;
	sf_AC_Frequency :REAL;
	sf_Apparent_Power :REAL;
	sf_Reactive_Power :REAL;
	sf_PowerFactor :REAL;
	sf_AC_Energy :REAL;
	sf_DC_Power :REAL;
	sf_Temperature :REAL;
	
END_VAR

ID := Data_Inverter[1];
Length := Data_Inverter[2];

sf_AC_Current	:= TO_REAL(EXPT(10,  Data_Inverter[7]));
sf_AC_Voltage	:= TO_REAL(EXPT(10, Data_Inverter[14]));
sf_AC_Power	:= TO_REAL(EXPT(10, Data_Inverter[16]));
sf_AC_Frequency	:= TO_REAL(EXPT(10, Data_Inverter[18]));
sf_Apparent_Power	:= TO_REAL(EXPT(10, Data_Inverter[20]));
sf_Reactive_Power	:= TO_REAL(EXPT(10, Data_Inverter[22]));
sf_PowerFactor	:= TO_REAL(EXPT(10, Data_Inverter[24]));
sf_AC_Energy	:= TO_REAL(EXPT(10, Data_Inverter[27]));
sf_DC_Power	:= TO_REAL(EXPT(10, Data_Inverter[33]));
sf_Temperature	:= TO_REAL(EXPT(10, Data_Inverter[38]));

AC_Current := Data_Inverter[3]*sf_AC_Current;
Phase_A_Current := Data_Inverter[4]*sf_AC_Current;
Phase_B_Current := Data_Inverter[5]*sf_AC_Current;
Phase_C_Current := Data_Inverter[6]*sf_AC_Current;

Phase_Voltage_AB := Data_Inverter[8]*sf_AC_Voltage;
Phase_Voltage_BC := Data_Inverter[9]*sf_AC_Voltage;
Phase_Voltage_CA := Data_Inverter[10]*sf_AC_Voltage;
Phase_Voltage_AN := Data_Inverter[11]*sf_AC_Voltage;
Phase_Voltage_BN := Data_Inverter[12]*sf_AC_Voltage;
Phase_Voltage_CN := Data_Inverter[13]*sf_AC_Voltage;

AC_Power := Data_Inverter[15]*sf_AC_Power;
AC_Frequency := TO_UINT(Data_Inverter[17]) *sf_AC_Frequency;
AC_Apparent_Power := Data_Inverter[19]*sf_Apparent_Power; 
AC_Reactive_Power := Data_Inverter[21] *sf_Reactive_Power;
AC_PowerFactor := Data_Inverter[23]*sf_PowerFactor;
//AC_Energy := (TO_WORD((Data_Inverter[25]) * EXPT(2,16)) + TO_WORD(Data_Inverter[26]))*sf_AC_Energy;
AC_Energy :=  TO_WORD(Data_Inverter[26])*sf_AC_Energy;
	
DC_Power := Data_Inverter[32] *sf_DC_Power;
Temperature := Data_Inverter[34] *sf_Temperature;
Status := Data_Inverter[39];
CASE Status OF
	1: State_Code := 'Aus';
	2: State_Code := 'Standby';
	3: State_Code := 'Startet';
	4: State_Code := 'Arbeitet';
	5: State_Code := 'LeistungRSeduktion';
	6: State_Code := 'Schaltet ab';
	7: State_Code := 'Fehler';
	8: State_Code := '';
	ELSE State_Code := 'N/A';
END_CASE

END_FUNCTION_BLOCK

// SunSpec_Translator/SunSpec_Model_Settings
FUNCTION_BLOCK SunSpec_Model_Settings
VAR_INPUT
	Data_Settings : ARRAY [1..30] OF INT;
END_VAR
VAR_OUTPUT
	ModelIdentifier              :INT;
    ModelLength                  :INT;
    MaximumPowerOutput           :REAL;
    VoltageAtPCC                 :REAL;
//     OffsetFromPCCToInverter      :REAL;
//     MaximumVoltage               :REAL;
//     MinimumVoltage               :REAL;
//     MaximumApparentPower         :REAL;
//     MaximumReactivePowerQ1       :REAL;
//     MaximumReactivePowerQ2       :REAL;
//     MaximumReactivePowerQ3       :REAL;
//     MaximumReactivePowerQ4       :REAL;
//     RampRateOfChangeOfActivePower:REAL;
//     MinimumPowerFactorQ1         :REAL;
//     MinimumPowerFactorQ2         :REAL;
//     MinimumPowerFactorQ3         :REAL;
//     MinimumPowerFactorQ4         :REAL;
END_VAR

VAR
    ScaleFactorMaximumPower          :REAL;
    ScaleFactorVoltageAtPCC          :REAL;
    ScaleFactorOffsetVoltage         :REAL;
    ScaleFactorMaximumVoltage        :REAL;
    ScaleFactorMinimumVoltage        :REAL;
    ScaleFactorMaximumApparentPower  :REAL;
    ScaleFactorMaximumReactivePower  :REAL;
    ScaleFactorRampRateOfChange      :REAL;
    ScaleFactorMinimumPowerFactor    :REAL;
END_VAR

ModelIdentifier := Data_Settings[1];
ModelLength := Data_Settings[2];

ScaleFactorMaximumPower         := EXPT(10, Data_Settings[23]);
ScaleFactorVoltageAtPCC         := EXPT(10, Data_Settings[24]);
// ScaleFactorOffsetVoltage        := EXPT(10, Data_Settings[25]);
// ScaleFactorMaximumVoltage       := EXPT(10, Data_Settings[26]);
// ScaleFactorMinimumVoltage       := EXPT(10, Data_Settings[26]);
// ScaleFactorMaximumApparentPower := EXPT(10, Data_Settings[27]);
// ScaleFactorMaximumReactivePower := EXPT(10, Data_Settings[28]);
// ScaleFactorRampRateOfChange     := EXPT(10, Data_Settings[29]);
// ScaleFactorMinimumPowerFactor   := EXPT(10, Data_Settings[30]);

MaximumPowerOutput := Data_Settings[3] * ScaleFactorMaximumPower;
VoltageAtPCC := Data_Settings[4] * ScaleFactorVoltageAtPCC;
// OffsetFromPCCToInverter := Data_Settings[5] * ScaleFactorOffsetVoltage;
// //MaximumVoltage := Data_Settings[6] * ScaleFactorMaximumVoltage;
// //MinimumVoltage := Data_Settings[7] * ScaleFactorMinimumVoltage;
// MaximumApparentPower := Data_Settings[8] * ScaleFactorMaximumApparentPower;
// MaximumReactivePowerQ1 := Data_Settings[9] * ScaleFactorMaximumReactivePower;
// MaximumReactivePowerQ2 := Data_Settings[10] * ScaleFactorMaximumReactivePower;
// MaximumReactivePowerQ3 := Data_Settings[11] * ScaleFactorMaximumReactivePower;
// MaximumReactivePowerQ4 := Data_Settings[12] * ScaleFactorMaximumReactivePower;
// //RampRateOfChangeOfActivePower := Data_Settings[13] * ScaleFactorRampRateOfChange;
// MinimumPowerFactorQ1 := Data_Settings[14] * ScaleFactorMinimumPowerFactor;
// MinimumPowerFactorQ2 := Data_Settings[15] * ScaleFactorMinimumPowerFactor;
// MinimumPowerFactorQ3 := Data_Settings[16] * ScaleFactorMinimumPowerFactor;
// MinimumPowerFactorQ4 := Data_Settings[17] * ScaleFactorMinimumPowerFactor;

END_FUNCTION_BLOCK

// SunSpec_Translator/SunSpec_Model_Status
FUNCTION_BLOCK SunSpec_Model_Status
VAR_INPUT
    Data_Status :ARRAY [1..50] OF INT; // Eingabedaten für Statusdaten
END_VAR
VAR_OUTPUT
    ModelIdentifier            :INT;
    ModelLength                :INT;
    PVInverterConnectionStatus :STRING;
    StorageInverterConnectionStatus :STRING;
    ECPConnectionStatus        :INT;
	AccumulatedACRealEnergyOutput :REAL;
//     AccumulatedACApparentEnergyOutput :REAL;
//     AccumulatedACReactiveEnergyQ1 :REAL;
//     AccumulatedACReactiveEnergyQ2 :REAL;
//     AccumulatedACReactiveEnergyQ3 :REAL;
//     AccumulatedACReactiveEnergyQ4 :REAL;
//     AvailableVARs              :INT;
//     AvailableWatts             :INT;
//     SetpointLimitStatus        :INT;
    ActiveControlStatus        :INT;
    SecondsSince2000           :DWORD;
//     RideThroughStatus          :INT;
    IsolationResistance        :REAL;
END_VAR
VAR
	ConnectionPV		:INT;
	ConnectionBat		:INT;
END_VAR

ModelIdentifier := Data_Status[1];
ModelLength := Data_Status[2];

ConnectionPV := Data_Status[3];
CASE ConnectionPV OF
	0: PVInverterConnectionStatus := 'Verbunden';
	1: PVInverterConnectionStatus := 'Bereit';
	2: PVInverterConnectionStatus := 'Arbeitet';
	ELSE PVInverterConnectionStatus := 'Nicht verbunden';
END_CASE

ConnectionBat := Data_Status[4];
CASE ConnectionBat OF
	0: StorageInverterConnectionStatus := 'Verbunden';
	1: StorageInverterConnectionStatus := 'Bereit';
	2: StorageInverterConnectionStatus := 'Arbeitet';
	ELSE PVInverterConnectionStatus := 'Nicht verbunden';
END_CASE
ECPConnectionStatus := Data_Status[5];

AccumulatedACRealEnergyOutput := TO_REAL(Data_Status[6]) + TO_REAL(Data_Status[7] * EXPT(2,32));
// AccumulatedACApparentEnergyOutput := TO_REAL(Data_Status[10]) + TO_REAL(Data_Status[11] * EXPT(2,32));
// AccumulatedACReactiveEnergyQ1 := TO_REAL(Data_Status[14]) + TO_REAL(Data_Status[15] * EXPT(2,32));
// AccumulatedACReactiveEnergyQ2 := TO_REAL(Data_Status[18]) + TO_REAL(Data_Status[19] * EXPT(2,32));
// AccumulatedACReactiveEnergyQ3 := TO_REAL(Data_Status[22]) + TO_REAL(Data_Status[23] * EXPT(2,32));
// AccumulatedACReactiveEnergyQ4 := TO_REAL(Data_Status[26]) + TO_REAL(Data_Status[27] * EXPT(2,32));
// 
// AvailableVARs := Data_Status[30];
// AvailableWatts := Data_Status[32];
// 
// SetpointLimitStatus := Data_Status[34];
ActiveControlStatus := Data_Status[36];



SecondsSince2000 := TO_DWORD(Data_Status[42]) + TO_DWORD(Data_Status[43] * EXPT(2,32));
// RideThroughStatus := Data_Status[44];

IsolationResistance := TO_REAL(Data_Status[45]) * EXPT(10, -Data_Status[46]);

END_FUNCTION_BLOCK

// SunSpec_Translator/SunSpec_Model_Controls
FUNCTION_BLOCK SunSpec_Model_Controls
VAR_INPUT
    Data_Controls :ARRAY [1..30] OF INT;
END_VAR
VAR_OUTPUT
    ModelIdentifier            :INT;
    ModelLength                :INT;
    ConnectionTimeWindow       :REAL;
    ConnectionTimeoutPeriod    :REAL;
    ConnectionControl          :STRING;
    PowerOutputPercent         :REAL;
    PowerOutputTimeWindow      :REAL;
    PowerOutputTimeoutPeriod   :REAL;
    PowerOutputRampTime        :REAL;
    PowerOutputEnable          :STRING;
    PowerFactorSetpoint        :REAL;
    PowerFactorTimeWindow      :REAL;
    PowerFactorTimeoutPeriod   :REAL;
    PowerFactorRampTime        :REAL;
    PowerFactorEnable          :INT;
    ReactivePowerMaxPercent    :REAL;
    ReactivePowerTimeWindow    :REAL;
    ReactivePowerTimeoutPeriod :REAL;
    ReactivePowerRampTime      :REAL;
    ReactivePowerLimitMode     :INT;
    ReactivePowerEnable        :INT;
END_VAR

VAR
    ScaleFactorPowerOutputPercent   :REAL;
    ScaleFactorPowerFactor          :REAL;
    ScaleFactorReactivePowerPercent :REAL;
	Connection		:INT;
	Throttle		:INT;
END_VAR

ModelIdentifier := Data_Controls[1];
ModelLength := Data_Controls[2];

ScaleFactorPowerOutputPercent := EXPT(10, Data_Controls[24]);
ScaleFactorPowerFactor := EXPT(10, Data_Controls[25]);
ScaleFactorReactivePowerPercent := EXPT(10, Data_Controls[26]);

ConnectionTimeWindow := TO_REAL(Data_Controls[3]);
ConnectionTimeoutPeriod := TO_REAL(Data_Controls[4]);

Connection := Data_Controls[5];
CASE Connection OF
	0: ConnectionControl := 'Standby';
	1: ConnectionControl := 'Ein';
	ELSE ConnectionControl := 'Nicht verbunden';
END_CASE

PowerOutputPercent := TO_REAL(Data_Controls[6]) * ScaleFactorPowerOutputPercent;
PowerOutputTimeWindow := TO_REAL(Data_Controls[7]);
PowerOutputTimeoutPeriod := TO_REAL(Data_Controls[8]);
PowerOutputRampTime := TO_REAL(Data_Controls[9]);

Throttle := Data_Controls[10];
CASE Throttle OF
	0: PowerOutputEnable := 'Aus';
	1: PowerOutputEnable := 'Ein';
	ELSE PowerOutputEnable := 'N/A';
END_CASE

PowerFactorSetpoint := TO_REAL(Data_Controls[11]) * ScaleFactorPowerFactor;
PowerFactorTimeWindow := TO_REAL(Data_Controls[12]);
PowerFactorTimeoutPeriod := TO_REAL(Data_Controls[13]);
PowerFactorRampTime := TO_REAL(Data_Controls[14]);
PowerFactorEnable := Data_Controls[15];

//ReactivePowerWMaxPercent := TO_REAL(Data_Controls[16]) * ScaleFactorReactivePowerPercent;
ReactivePowerMaxPercent := TO_REAL(Data_Controls[17]) * ScaleFactorReactivePowerPercent;
//ReactivePowerAvailablePercent := TO_REAL(Data_Controls[18]) * ScaleFactorReactivePowerPercent;

ReactivePowerTimeWindow := TO_REAL(Data_Controls[19]);
ReactivePowerTimeoutPeriod := TO_REAL(Data_Controls[20]);
ReactivePowerRampTime := TO_REAL(Data_Controls[21]);

ReactivePowerLimitMode := Data_Controls[22];
ReactivePowerEnable := Data_Controls[23];

END_FUNCTION_BLOCK

// SunSpec_Translator/SunSpec_Model_MPPT
FUNCTION_BLOCK SunSpec_Model_MPPT
VAR_INPUT
    Data_MPPT :ARRAY [1..30] OF INT;
END_VAR
VAR_OUTPUT
    ModelIdentifier            :INT;
    ModelLength                :INT;
//     GlobalEvents               :INT;
    NumberOfModules            :INT;
//     TimestampPeriod            :INT;
    ModuleID                   :INT;
    ModuleIDString             :STRING;
    DCCurrent                  :REAL;
    DCVoltage                  :REAL;
    DCPower                    :REAL;
    LifetimeEnergy             :REAL;
    Timestamp                  :DWORD;
END_VAR

VAR
    ScaleFactorDCA    :REAL;
    ScaleFactorDCV    :REAL;
    ScaleFactorDCW    :REAL;
    ScaleFactorDCWH   :REAL;
END_VAR

ModelIdentifier := Data_MPPT[1];
ModelLength := Data_MPPT[2];

ScaleFactorDCA := EXPT(10, Data_MPPT[3]);
ScaleFactorDCV := EXPT(10, Data_MPPT[4]);
ScaleFactorDCW := EXPT(10, Data_MPPT[5]);
ScaleFactorDCWH := EXPT(10, Data_MPPT[6]);

//GlobalEvents := Data_MPPT[7];
NumberOfModules := Data_MPPT[9];
//TimestampPeriod := Data_MPPT[10];

ModuleID := Data_MPPT[11];
ModuleIDString := 'MPPT 1';

DCCurrent := TO_REAL(TO_UINT(Data_MPPT[20])) * ScaleFactorDCA;
DCVoltage := TO_REAL(TO_UINT(Data_MPPT[21])) * ScaleFactorDCV;
DCPower := TO_REAL(TO_UINT(Data_MPPT[22])) * ScaleFactorDCW;

LifetimeEnergy := TO_REAL((TO_WORD(Data_MPPT[23]) * EXPT(2,16)) + TO_WORD(Data_MPPT[24])) * ScaleFactorDCWH;
Timestamp := TO_DWORD((Data_MPPT[25] * EXPT(2,16)) + Data_MPPT[26]);

END_FUNCTION_BLOCK

// SunSpec_Translator/SunSpec_Model_Meter
FUNCTION_BLOCK SunSpec_Model_Meter
VAR_INPUT
    Data_Meter :ARRAY [1..75] OF INT;
END_VAR
VAR_OUTPUT
    ModelIdentifier            :INT;
    ModelLength                :INT;
    TotalACCurrent             :REAL;
    PhaseACurrentA             :REAL;
    PhaseACurrentB             :REAL;
    PhaseACurrentC             :REAL;
    LineToNeutralVoltage       :REAL;
    PhaseVoltageAN             :REAL;
    PhaseVoltageBN             :REAL;
    PhaseVoltageCN             :REAL;
    LineToLineVoltage          :REAL;
    PhaseVoltageAB             :REAL;
    PhaseVoltageBC             :REAL;
    PhaseVoltageCA             :REAL;
    Frequency                  :REAL;
    TotalRealPower             :REAL;
    WattsPhaseA                :REAL;
    WattsPhaseB                :REAL;
    WattsPhaseC                :REAL;
    ACApparentPower            :REAL;
    VAPhaseA                   :REAL;
    VAPhaseB                   :REAL;
    VAPhaseC                   :REAL;
    TotalReactivePower         :REAL;
    VARPhaseA                  :REAL;
    VARPhaseB                  :REAL;
    VARPhaseC                  :REAL;
    PowerFactor                :REAL;
    PowerFactorPhaseA          :REAL;
    PowerFactorPhaseB          :REAL;
    PowerFactorPhaseC          :REAL;
    TotalRealEnergyExported    :REAL;
    TotalRealEnergyImported    :REAL;
    TotalApparentEnergyExported:REAL;
    TotalApparentEnergyImported:REAL;
END_VAR

VAR
    ScaleFactorCurrent         :REAL;
    ScaleFactorVoltage         :REAL;
    ScaleFactorFrequency       :REAL;
    ScaleFactorPower           :REAL;
    ScaleFactorEnergy          :REAL;
    ScaleFactorApparentPower   :REAL;
    ScaleFactorReactivePower   :REAL;
    ScaleFactorPowerFactor     :REAL;
	
	 dwTemp : DWORD;
    diTemp : DINT;
END_VAR

ModelIdentifier := Data_Meter[1];
ModelLength := Data_Meter[2];
ScaleFactorCurrent := EXPT(10, Data_Meter[7]);
ScaleFactorVoltage := EXPT(10, Data_Meter[16]);
ScaleFactorFrequency := EXPT(10, Data_Meter[18]);
ScaleFactorPower := EXPT(10, Data_Meter[23]);
ScaleFactorEnergy := EXPT(10, Data_Meter[55]);
ScaleFactorApparentPower := EXPT(10, Data_Meter[28]);
ScaleFactorReactivePower := EXPT(10, Data_Meter[33]);
ScaleFactorPowerFactor := EXPT(10, Data_Meter[38]);

TotalACCurrent := TO_REAL(Data_Meter[3]) * ScaleFactorCurrent;
PhaseACurrentA := TO_REAL(Data_Meter[4]) * ScaleFactorCurrent;
PhaseACurrentB := TO_REAL(Data_Meter[5]) * ScaleFactorCurrent;
PhaseACurrentC := TO_REAL(Data_Meter[6]) * ScaleFactorCurrent;
LineToNeutralVoltage := TO_REAL(Data_Meter[8]) * ScaleFactorVoltage;
PhaseVoltageAN := TO_REAL(Data_Meter[9]) * ScaleFactorVoltage;
PhaseVoltageBN := TO_REAL(Data_Meter[10]) * ScaleFactorVoltage;
PhaseVoltageCN := TO_REAL(Data_Meter[11]) * ScaleFactorVoltage;
LineToLineVoltage := TO_REAL(Data_Meter[12]) * ScaleFactorVoltage;
PhaseVoltageAB := TO_REAL(Data_Meter[13]) * ScaleFactorVoltage;
PhaseVoltageBC := TO_REAL(Data_Meter[14]) * ScaleFactorVoltage;
PhaseVoltageCA := TO_REAL(Data_Meter[15]) * ScaleFactorVoltage;
Frequency := TO_REAL(Data_Meter[17]) * ScaleFactorFrequency;
TotalRealPower := TO_REAL(Data_Meter[19]) * ScaleFactorPower;
WattsPhaseA := TO_REAL(Data_Meter[20]) * ScaleFactorPower;
WattsPhaseB := TO_REAL(Data_Meter[21]) * ScaleFactorPower;
WattsPhaseC := TO_REAL(Data_Meter[22]) * ScaleFactorPower;
ACApparentPower := TO_REAL(Data_Meter[24]) * ScaleFactorApparentPower;
VAPhaseA := TO_REAL(Data_Meter[25]) * ScaleFactorApparentPower;
VAPhaseB := TO_REAL(Data_Meter[26]) * ScaleFactorApparentPower;
VAPhaseC := TO_REAL(Data_Meter[27]) * ScaleFactorApparentPower;
TotalReactivePower := TO_REAL(Data_Meter[29]) * ScaleFactorReactivePower;
VARPhaseA := TO_REAL(Data_Meter[30]) * ScaleFactorReactivePower;
VARPhaseB := TO_REAL(Data_Meter[31]) * ScaleFactorReactivePower;
VARPhaseC := TO_REAL(Data_Meter[32]) * ScaleFactorReactivePower;
PowerFactor := TO_REAL(Data_Meter[34]) * ScaleFactorPowerFactor;
PowerFactorPhaseA := TO_REAL(Data_Meter[35]) * ScaleFactorPowerFactor;
PowerFactorPhaseB := TO_REAL(Data_Meter[36]) * ScaleFactorPowerFactor;
PowerFactorPhaseC := TO_REAL(Data_Meter[37]) * ScaleFactorPowerFactor;
TotalRealEnergyExported := TO_REAL(Data_Meter[39]) * ScaleFactorEnergy;
TotalRealEnergyImported := TO_REAL(Data_Meter[40]) * ScaleFactorEnergy;
TotalApparentEnergyExported := TO_REAL(Data_Meter[42]) * ScaleFactorApparentPower;
TotalApparentEnergyImported := TO_REAL(Data_Meter[43]) * ScaleFactorApparentPower;


(*
ModelIdentifier := Data_Meter[1];
ModelLength := Data_Meter[2];

ScaleFactorCurrent := 0.001;
ScaleFactorVoltage := 0.1;
ScaleFactorFrequency := 0.01;
ScaleFactorPower := 0.001;
ScaleFactorEnergy := 0.01;
ScaleFactorApparentPower := 0.01;
ScaleFactorReactivePower := 0.01;
ScaleFactorPowerFactor := 0.01;

TotalACCurrent := TO_REAL(Data_Meter[3]) * ScaleFactorCurrent;
PhaseACurrentA := TO_REAL(Data_Meter[4]) * ScaleFactorCurrent;
PhaseACurrentB := TO_REAL(Data_Meter[5]) * ScaleFactorCurrent;
PhaseACurrentC := TO_REAL(Data_Meter[6]) * ScaleFactorCurrent;
LineToNeutralVoltage := TO_REAL(Data_Meter[7]) * ScaleFactorVoltage;
PhaseVoltageAN := TO_REAL(Data_Meter[8]) * ScaleFactorVoltage;
PhaseVoltageBN := TO_REAL(Data_Meter[9]) * ScaleFactorVoltage;
PhaseVoltageCN := TO_REAL(Data_Meter[10]) * ScaleFactorVoltage;
LineToLineVoltage := TO_REAL(Data_Meter[11]) * ScaleFactorVoltage;
PhaseVoltageAB := TO_REAL(Data_Meter[12]) * ScaleFactorVoltage;
PhaseVoltageBC := TO_REAL(Data_Meter[13]) * ScaleFactorVoltage;
PhaseVoltageCA := TO_REAL(Data_Meter[14]) * ScaleFactorVoltage;
Frequency := TO_REAL(Data_Meter[17]) * ScaleFactorFrequency;
TotalRealPower := TO_REAL(Data_Meter[16]) * ScaleFactorPower;
WattsPhaseA := TO_REAL(Data_Meter[17]) * ScaleFactorPower;
WattsPhaseB := TO_REAL(Data_Meter[18]) * ScaleFactorPower;
WattsPhaseC := TO_REAL(Data_Meter[19]) * ScaleFactorPower;
ACApparentPower := TO_REAL(Data_Meter[20]) * ScaleFactorApparentPower;
VAPhaseA := TO_REAL(Data_Meter[21]) * ScaleFactorApparentPower;
VAPhaseB := TO_REAL(Data_Meter[22]) * ScaleFactorApparentPower;
VAPhaseC := TO_REAL(Data_Meter[23]) * ScaleFactorApparentPower;
TotalReactivePower := TO_REAL(Data_Meter[24]) * ScaleFactorReactivePower;
VARPhaseA := TO_REAL(Data_Meter[25]) * ScaleFactorReactivePower;
VARPhaseB := TO_REAL(Data_Meter[26]) * ScaleFactorReactivePower;
VARPhaseC := TO_REAL(Data_Meter[27]) * ScaleFactorReactivePower;
PowerFactor := TO_REAL(Data_Meter[28]) * ScaleFactorPowerFactor;
PowerFactorPhaseA := TO_REAL(Data_Meter[29]) * ScaleFactorPowerFactor;
PowerFactorPhaseB := TO_REAL(Data_Meter[30]) * ScaleFactorPowerFactor;
PowerFactorPhaseC := TO_REAL(Data_Meter[31]) * ScaleFactorPowerFactor;
TotalRealEnergyExported := TO_REAL(Data_Meter[32]) * ScaleFactorEnergy;
TotalRealEnergyImported := TO_REAL(Data_Meter[33]) * ScaleFactorEnergy;
TotalApparentEnergyExported := TO_REAL(Data_Meter[34]) * ScaleFactorApparentPower;
TotalApparentEnergyImported := TO_REAL(Data_Meter[35]) * ScaleFactorApparentPower;
*)

END_FUNCTION_BLOCK

// Inverter
PROGRAM Inverter
VAR
	
	MPPT_initialisiert 		:BOOL :=FALSE;					// Flag
	
	zielLeistung			:REAL;							// Einzustellende Leistung [W]
	zielLeistungProzent 	:REAL;							// Einzustellende Leistung [%]
	abweichungLeistung		:REAL;							// Abeichung zwischen eingestellter und effektiver Leistung
	
	initialLeistungProzent 	:UINT; 							// Mit welcher Leistung gestartet wird [%]
	effektivLeistung		:REAL; 							// Aktuelle Inverterleistung [W]
	toleranzLeistung		:REAL; 							// Erlaubte Abweichung, damit es als erreicht gilt [W]
	anpassungLeistung		:REAL; 							// Leistungsanpassungsschritt [%]
	
	
	TimerMPPT				:TON;
	TimerTimeout			:TON;
	intervallMPPT			:TIME;							// Wie lange gewartet wird, bis MPP einen nächsten Schritt macht [s]
	intervallTimeout		:TIME;							// Wie lange, bis die Leistung als  nicht erreicht betrachtet wird [s]
	
	effektivDrehzahl		:REAL;							// Verwendete Drehzahl für MPPT [rpm]
  	toleranzDrehzahl		:REAL;							// Angenommene Ungenauigkeit [rpm]
	sollDrehzahl			:INT;							// Sollwert für Drehzahlregulierung [rpm]
	
	
	TimerHerunterfahren	:TON;
	intervallHerunterfahren	:TIME;							// Wie lange zwischen den Schritten gewartet wird [s]


	diff: REAL;
END_VAR

(* Allgemeines -------------------------------------------------------------------------------------------------*)
// Setzen der Parameter
GV.inv_IP := GV.p_Inverter_IP;
initialLeistungProzent := GV.p_Leistung_Init;
effektivLeistung := GV.r_LeistungAC;
toleranzLeistung := GV.p_Leistung_Toleranz;
anpassungLeistung := GV.p_Leistung_Anpassung;
intervallMPPT := GV.p_MPPT_Intervall;
intervallTimeout := GV.p_MPPT_Timeout;
effektivDrehzahl := GV.sys_Drehzahl;
toleranzDrehzahl := GV.p_Drehzahl_Toleranz;
sollDrehzahl := GV.p_Drehzahl_soll;
intervallHerunterfahren := GV.p_Herunterfahren_Intervall;


// Drehzahldifferenz berechnen
diff := ABS(GV.sys_Drehzahl - GV.p_Drehzahl_soll);

// Abstufung MPPT
IF diff > GV.p_Drehzahl_Toleranz * 5 THEN
    anpassungLeistung := GV.p_Leistung_Anpassung * 5;
	intervallMPPT := GV.p_MPPT_Intervall/3;
ELSIF diff > GV.p_Drehzahl_Toleranz * 3 THEN
   
	intervallMPPT := GV.p_MPPT_Intervall* 2;
ELSIF diff > GV.p_Drehzahl_Toleranz * 1 THEN
    anpassungLeistung := GV.p_Leistung_Anpassung * 1.5;
	
ELSE
    anpassungLeistung := GV.p_Leistung_Anpassung * 1.0;
	intervallMPPT := GV.p_MPPT_Intervall;
END_IF


(*__________________________________                                                                      *)

// Abfrage ob Inverter erfolgreich kommuniziert 
IF GV.r_SpannungPCC >0 AND NOT (GV.stoerung_Modbus_Lesen OR GV.stoerung_Modbus_Schreiben) THEN
	GV.inv_ein := TRUE;
ELSE GV.inv_ein := FALSE;
END_IF


(*__________________________________                                                                      *)

// Inverterzustände
IF GV.r_StateCode = 'Arbeitet' THEN
	GV.inv_bereit :=TRUE;
ELSE GV.inv_bereit :=FALSE;
END_IF
IF GV.r_StateCode = 'Standby' THEN
	GV.inv_standby := TRUE;
ELSE
	GV.inv_standby := FALSE;
END_IF
// --

IF GV.r_LeistungAC < 20 THEN
	GV.inv_betrieb := FALSE;
	
ELSE GV.inv_betrieb := TRUE;	
	GV.inv_leerlauf := FALSE;
END_IF


(*__________________________________                                                                      *)

(* Steuerung ---------------------------------------------------------------------------------------------*)

// Inverter in Leerlauf

IF GV.inv_leerlauf THEN
	 GV.sys_LeistungBegrenzung := TO_UINT(0); // Leerlauf: Stellt sicher, dass nicht produziert wird
	 zielLeistungProzent := 0;;
END_IF


(*__________________________________                                                                      *)


// Berechnungen für einfachere Handhabung 
zielLeistung := zielLeistungProzent * 3000 / 10000;  // Auf Inverter mit 3000W maximalleistung festgelegt
abweichungLeistung := ABS(effektivLeistung - zielLeistung);

(*__________________________________                                                                      *)

// Begrenzt die Variable auf gültige Werte (0 - 100.00 %)
IF zielLeistungProzent < 0 THEN
    zielLeistungProzent := 0;
ELSIF zielLeistungProzent > 10000 THEN
    zielLeistungProzent := 10000;
END_IF


// Rückstellen der Leistung
IF GV.sys_aus OR GV.sys_start OR GV.sys_bereit THEN
	zielLeistungProzent := 0;
END_IF

(*__________________________________                                                                      *)

// MPPT
IF GV.sys_MPPT_aktiv THEN
GV.inv_leerlauf := FALSE;	
	// MPPT starten	
    IF NOT MPPT_initialisiert THEN
        GV.sys_LeistungBegrenzung := TO_UINT(initialLeistungProzent); 
		TimerMPPT(IN:=FALSE);
		MPPT_initialisiert := TRUE;    
        	// Warten bis Leistung erreicht wird
    ELSE
        IF TimerMPPT.Q THEN	
		// MPPT macht den nächsten Schritt
				
           IF effektivDrehzahl > sollDrehzahl  + toleranzDrehzahl THEN
                zielLeistungProzent := zielLeistungProzent + anpassungLeistung;
				GV.sys_MPP_erreicht := FALSE;
			ELSE
				
				IF 	effektivDrehzahl < sollDrehzahl  - toleranzDrehzahl THEN
					zielLeistungProzent := zielLeistungProzent - anpassungLeistung;
					GV.sys_MPP_erreicht := FALSE;
				ELSE
					GV.sys_MPP_erreicht := TRUE;
				END_IF	
            END_IF
			
            GV.sys_LeistungBegrenzung := TO_UINT(zielLeistungProzent);
            TimerMPPT(IN:=FALSE);
			// Warten bis die Leistung erreicht wird
        END_IF
     END_IF   
	
    // Überprüfung, ob die gewünschte Leistung erreicht wird
        IF ABS(abweichungLeistung) <= ABS(toleranzLeistung) THEN
            MPPT_initialisiert := TRUE;
            TimerMPPT(IN:=TRUE, PT:= intervallMPPT);
			TimerTimeout(IN:=FALSE);    
		ELSE
			TimerTimeout(IN:=TRUE, PT:= intervallTimeout);   
        END_IF
		    
    	// Wird die eingestellte Leistung nicht erreicht, wurde der MPP überschritten.  
        IF TimerTimeout.Q THEN
            zielLeistungProzent := zielLeistungProzent - anpassungLeistung;
            GV.sys_LeistungBegrenzung := TO_UINT(zielLeistungProzent);
            TimerTimeout(IN:=FALSE);
        END_IF
    
ELSE
	MPPT_initialisiert := FALSE;
	GV.sys_MPP_erreicht := FALSE;
END_IF

(*__________________________________                                                                      *)

// Inverter herunterfahren
IF GV.sys_herunterfahren THEN
	GV.sys_MPPT_aktiv := FALSE;
	TimerHerunterfahren(IN:=TRUE,PT:=intervallHerunterfahren);
	
	IF effektivLeistung < toleranzLeistung THEN
		TimerHerunterfahren(IN:=FALSE);
		GV.sys_LeistungBegrenzung := TO_UINT(0); // Leerlauf: Stellt sicher, dass nicht produziert wird
	 	zielLeistungProzent := 0;	
		GV.inv_leerlauf := TRUE;	
	
		
		
	END_IF
ELSE
	TimerHerunterfahren(IN:=FALSE);	
END_IF

IF TimerHerunterfahren.Q THEN
		zielLeistungProzent := zielLeistungProzent - anpassungLeistung;
		GV.sys_LeistungBegrenzung := TO_UINT(zielLeistungProzent);
		TimerHerunterfahren(IN:=FALSE);
END_IF

(*__________________________________                                                                      *)

END_PROGRAM

// Berechnungen
PROGRAM Berechnungen
VAR
	U_s		 	:REAL;			 	// Strangspannung [V]
	U_p 		:REAL;  			// Polradspannung [V]
	I_s 		:REAL;				// Strangstrom [A]
	f_el 		:REAL; 				// Elektrische Drehzahl [Hz]
	N_est 		:REAL; 				// angenommene Drehzahl [rpm]
	N_calc 		:REAL; 				// berechnete Drehzahl [rpm]
	X_d			:REAL;				// Statorreaktanz [Ohm]
	R_s 		:REAL := 4; 		// Statorwiderstand [Ohm]
	L_d 		:REAL := 0.0186; 	// Statorinduktivität [H]
	c_volt_rpm	:REAL := 0.865321215; 	// Faktor Volt / rpm
	c_hertz_rpm	:REAL := 0.083476386; 	// Faktor Hetz / rpm
	c_U_ac_dc	:REAL := 1.31; 			// Faktor Gleichrichter Spannung AC zu DC
	n_Getriebe	:REAL := 93.5;			// 	Übersetzungsverhältnis des Getriebes
	
	i			:INT;
	iteration	:INT := 5;				// Wie oft die Iteration ausgeführt werden soll
	
	
	ForwardCounter 		:OBIOForwardCounter;
    ImpulseProSekunde	:REAL;		// Anzahl der Impulse pro Sekunde
    ImpulsZaehler		:INT; 		// Zähler für die Impulse
    VergangeneZeit		:TIME; 		// Zeit seit dem letzten Reset des Zählers
    Zeitgeber: TON; 				// Zeitgeber zur Zeitmessung
    SensorEingang		:BOOL; 		// Eingangssignal vom Drehzahlsensor
	
	differenzCounter	:UDINT;
	vorherCounter		:UDINT;
	effektivCounter		:UDINT;

	
logger : FB_DataLogger;
aWerte : ARRAY[1..3] OF REAL;
	
	// Show
	P_Bilanz :REAL;
	LetzteZeit : TIME := T#0S;
	deltaT : REAL; // Zeit in Stunden
    deltaE : REAL; // Energie in Wh
	DrehzahlLogger : FB_MQTT_Logger;
	LeistungLogger : FB_MQTT_Logger;
END_VAR


(* Allgemeines ------------------------------------------------------------------------------------------- *)

// Berechnung der eingestellten Leistung
GV.inv_MaxLeistungEingestellt := GV.inv_MaxLeistungEingestellt * GV.r_LeistungBegrenzung / 100;

(*__________________________________   


                                                                   *)

(* Bestimmen der Drehzahl --------------------------------------------------------------------------------*)
(* Konstanten stammen aus dem Messprotokoll *)
(* Drehzahlberechnung über Maschinenparameter*)
U_s := GV.r_SpannungDC / c_U_ac_dc;		
I_s := GV.r_StromDC * 0.7785 + 0.0987;		

// Estimator der Drehzahl
N_est := U_s / c_volt_rpm;					
GV.sys_Drehzahl_Estimator := TO_UINT(N_est);

// Iterative Berechnung zur Verbesserung der Genauigkeit
FOR i := 1 TO iteration DO
	IF i = 1 THEN
		f_el := N_est * c_hertz_rpm;
	ELSE	
    	f_el := N_calc * c_hertz_rpm;
	END_IF
    X_d := 1 / (L_d * f_el);
    U_p := SQRT(EXPT(U_s + R_s * I_s, 2) + EXPT(I_s * X_d, 2));
    N_calc := U_p / c_volt_rpm;
END_FOR

GV.sys_Drehzahl_Rechner:= TO_UINT(N_calc);



(*__________________________________                                                                      *)


// Drehzahlberechnung über Sensor mittels Forward Counter

ForwardCounter(Enable := TRUE, Channel := 0, Set := TRUE, EnableLimit := FALSE);
GV.I_Counter := ForwardCounter.CounterValue;

// Zeitgeber-Einstellung
Zeitgeber(IN := TRUE, PT := T#2S);
IF Zeitgeber.Q THEN
    // Berechnung der Impulse pro Sekunde
    differenzCounter := GV.I_Counter - vorherCounter;
    
    // Berechnung der Drehzahl in RPM
    GV.sys_Drehzahl_Sensor := TO_REAL( differenzCounter )/ GV.p_Sensor_Impulse * 60 / 2;
    
    // Reset des Impulszählers und des Zeitgebers
    vorherCounter := GV.I_Counter;
    Zeitgeber(IN := FALSE);
END_IF

(*__________________________________                                                                      *)

// Systemdrehzahl setzen

IF  GV.O_Hauptschuetz THEN
	
	GV.sys_Drehzahl := GV.sys_Drehzahl_Rechner;	
ELSE
	GV.sys_Drehzahl := GV.sys_Drehzahl_Sensor;
END_IF


(*__________________________________                                                                      *)

(*  Visu -------------------------------------------------------------------------------------------------*)

// Manuelle Leistungsbegrenzung über Visu
IF GV.v_LeistungBegrenzung_ein THEN
	GV.w_LeistungBegrenzung := TO_UINT(TO_REAL(GV.v_LeistungBegrenzung) * 10000 / 3000) ;

ELSE GV.w_LeistungBegrenzung := GV.sys_LeistungBegrenzung;
END_IF

(*__________________________________                                                                      *)

// Drehzahlberechnung des Wasserrads
GV.sys_Drehzahl_Wasserrad := GV.sys_Drehzahl / n_Getriebe;

(*__________________________________                                                                      *)

// Bestimmern, ob Generator dreht

IF GV.sys_Drehzahl > 0 THEN
	GV.v_Geni_lauft :=TRUE;
ELSE 
	GV.v_Geni_lauft :=FALSE;	
END_IF

(*__________________________________                                                                      *)

// Werte ins Array packen
aWerte[1] := GV.p_Drehzahl_soll;
aWerte[2] := GV.sys_Drehzahl;
aWerte[3] := GV.r_LeistungAC;

// Datenlogger aufrufen
logger(
    xEnable := TRUE,
    rValues := aWerte
);


(*__________________________________                                                                      *)

// Virtueller Akku für Show
// === Berechnung Kaffeemaschine ===
GV.v_Kaffeemaschine := GV.r_LeistungAC + GV.r_sm_Leistung -15.0; // Verbrauch Steuerung
IF GV.v_Kaffeemaschine < 0.0 THEN
    GV.v_Kaffeemaschine := 0.0;
END_IF

// === Bilanz aus Produktion und Verbrauch ===
P_Bilanz := GV.r_LeistungAC - GV.v_Kaffeemaschine;

// === Zeitdifferenz in Stunden ===
deltaT := TO_REAL(TO_TIME(TIME()) - LetzteZeit) / 3600000.0;
LetzteZeit := TIME();

// === Änderung des Speicherinhalts ===
deltaE := P_Bilanz * deltaT;

IF GV.v_speicher_start THEN
    GV.v_Speicher := GV.v_Speicher + deltaE;

    // Begrenzen
    IF GV.v_Speicher > 300.0 THEN
        GV.v_Speicher := 300.0;
    ELSIF GV.v_Speicher < 0.0 THEN
        GV.v_Speicher := 0.0;
    END_IF
END_IF


// MQTT Logger

(* DrehzahlLogger(
    xEnable := TRUE,
    xTopic := 'Drehzahl',
	rData := GV.sys_Drehzahl
);
LeistungLogger(
    xEnable := TRUE,
    xTopic := 'Leistung',
	rData := GV.r_LeistungAC
);
*)

END_PROGRAM

// FB_DataLogger
FUNCTION_BLOCK FB_DataLogger
VAR_INPUT
    xEnable      : BOOL;
    rValues      : ARRAY[1..3] OF REAL; // Soll, Ist, Leistung
    tInterval    : TIME := T#5s;
END_VAR

VAR
    tonTrig      : TON;
	tRTC		:SYSTIME;
    tNow         : DT;
    tNowTime     : TIME;
    tStartTime   : TIME;
    bFirstCall   : BOOL := TRUE;

    iIndex       : INT := 1;
    
    aValues      : ARRAY[1..2000, 1..3] OF REAL;
    aTimeStamps  : ARRAY[1..2000] OF DT;
    aTimeSeconds : ARRAY[1..2000] OF REAL;

    // Visualisierungsfähige Arrays
    aDrehzahlSoll: ARRAY[1..2000] OF REAL;
    aDrehzahlIst : ARRAY[1..2000] OF REAL;
    aLeistung    : ARRAY[1..2000] OF REAL;
END_VAR

// Aktuellen Zeitstempel lesen

SysTimeRtcHighResGet(pTimestamp:= tRTC);
tNow := TO_DT(TO_INT(tRTC/1000));
tNowTime := DT_TO_TOD(tNow) - TOD#00:00:00;

// Einmalige Initialisierung
IF bFirstCall THEN
    tStartTime := tNowTime;
    bFirstCall := FALSE;
END_IF

// Intervall-Trigger
tonTrig(IN := xEnable, PT := tInterval);

IF tonTrig.Q AND xEnable THEN
    IF iIndex <= 2000 THEN
        // Werte speichern
        aValues[iIndex, 1] := rValues[1];
        aValues[iIndex, 2] := rValues[2];
		
        aValues[iIndex, 3] := rValues[3];

        // Zeit speichern
        aTimeStamps[iIndex] := tNow;

        // Sekundenzählung relativ zum Start
        aTimeSeconds[iIndex] := TO_REAL(TIME_TO_REAL(tNowTime - tStartTime)) / 1000.0;

        // Visualisierungsarrays befüllen
        aDrehzahlSoll[iIndex] := rValues[1];
        aDrehzahlIst[iIndex]  := rValues[2];
        aLeistung[iIndex]     := rValues[3];

        // Index hochzählen
        iIndex := iIndex + 1;
		tonTrig(IN:=FALSE);
	ELSE 
iIndex :=1;
    END_IF
END_IF

END_FUNCTION_BLOCK

// FB_MQTT_Logger
FUNCTION_BLOCK FB_MQTT_Logger
VAR_INPUT
    xEnable    : BOOL;         // Start/Stop
	xTopic		:STRING;		//Topicname
    rData	  : REAL;         // Sensorvalue
    
END_VAR

VAR_OUTPUT
    xConnected : BOOL;         // Verbindung aktiv
    xError     : BOOL;         // Fehler aufgetreten
    sError     : STRING(255);  // Fehlerbeschreibung
END_VAR

VAR
    fbClient     : MQTT.MQTTClient;
    fbPublish    : MQTT.MQTTPublish;

    sBrokerIP    : STRING(80) := '192.168.178.42';
    uiPort       : UINT := 1883;
    sClientID    : STRING(255) := 'SGSclient';

	 sTopic       : STRING(255) := 'SGS/logger';   // ASCII-safe
    wsTopic      : WSTRING(1024);
	sPayload		:STRING(255);
    wsPayload    : WSTRING(1024);

    abyPayload   : ARRAY[0..511] OF BYTE;
    udiPayloadSize : UDINT;

    tLastSend    : TIME := T#0s;
    tInterval    : TIME := T#5s;

    sDataValue : STRING(20);
    sLeistungStr : STRING(20);
END_VAR

sTopic := CONCAT('SGS/',xTopic);

wsTopic := TO_WSTRING(sTopic);

// Verbindung Client starten/stoppen
fbClient(
    xEnable := xEnable,
    sHostname := sBrokerIP,
    uiPort := uiPort,
    sClientId := sClientID
);

xConnected := fbClient.xConnectedToBroker;
xError := fbClient.xError;

IF xError THEN
    sError := CONCAT('MQTT Fehler: ', TO_STRING(fbClient.eMQTTError));
ELSE
    sError := '';
END_IF

// Nur senden wenn verbunden + Intervall eingehalten
IF xConnected AND (TIME() - tLastSend >= tInterval) THEN
    sDataValue := REAL_TO_STRING(rData);

	
sPayload := ''; // <--- Initialisierung sicherstellen
sPayload := CONCAT(sPayload, sDataValue);
wsPayload := TO_WSTRING(sPayload);


    udiPayloadSize := WSTRING_TO_BYTEARRAY_UTF8(wsPayload, ADR(abyPayload), SIZEOF(abyPayload));

    // Flanke erzeugen
    IF NOT fbPublish.xBusy AND NOT fbPublish.xDone THEN
        fbPublish.xExecute := TRUE;
    ELSE
        fbPublish.xExecute := FALSE;
    END_IF;

    // Publish
    fbPublish(
        xExecute := fbPublish.xExecute,
        mqttClient := fbClient,
        wsTopicName := wsTopic,
        eQoS := MQTT.MQTT_QOS.QoS0,
        xRetain := FALSE,
        xReDelivery := FALSE,
        pbPayload := ADR(abyPayload),
        udiPayloadSize := udiPayloadSize
    );

    tLastSend := TIME();
END_IF

END_FUNCTION_BLOCK

// WSTRING_TO_BYTEARRAY_UTF8
FUNCTION WSTRING_TO_BYTEARRAY_UTF8 : UINT
VAR_INPUT
    wsIn  : WSTRING(512);
    pDest : POINTER TO BYTE;
    uiMax : UINT;
END_VAR
VAR
    i     : UINT := 0;
    c     : BYTE;
END_VAR

FOR i := 0 TO uiMax - 1 DO
    c := TO_BYTE(wsIn[i]);
    IF c = 0 THEN
        EXIT;
    END_IF
    pDest[i] := c;
END_FOR

WSTRING_TO_BYTEARRAY_UTF8 := i;

END_FUNCTION

// Systemzustand
PROGRAM Systemzustand
VAR
	Systemzustand: INT;
	Busy: BOOL;
	
	ExecuteFlag: BOOL;
	Done: BOOL;
	TimerLadeschuetz :TON;
	
	TimerAuto :TON;
	BLINK_Starten: BLINK;
	BLINK_bereit: BLINK;
	BLINK_Stoerung: BLINK;
	Auto_ein: BOOL;
END_VAR

// Bedienknöpfe

GV.sys_Einschalten := GV.I_Einschalten OR GV.v_Einschalten;
GV.sys_Ausschalten := GV.I_Ausschalten OR GV.v_Ausschalten;

//Automatik einschalten mit 3s auf Ein
TimerAuto(IN := GV.sys_Einschalten, PT:= T#3S);

IF TimerAuto.Q THEN
	GV.p_Automatik := TRUE;
END_IF

IF GV.p_Automatik THEN
	Auto_ein := FALSE;
	// Einschaltbedingung Automatik
	IF GV.sys_Drehzahl >= GV.p_Drehzahl_min THEN
		Auto_ein := TRUE;
	END_IF
END_IF

//Automatik ausschalten 
IF GV.sys_Ausschalten THEN
	GV.p_Automatik := FALSE;
END_IF

// Störung überprüfen
IF GV.sammelstoerung THEN
	GV.O_Steuerspannung := FALSE;
	GV.p_Automatik := FALSE;
	Systemzustand := 0;
	
ELSE
// Störungsfrei	

IF NOT GV.inv_ein THEN
		Systemzustand := 0;
END_IF
	
IF GV.I_Notaus THEN
	GV.O_Steuerspannung:= FALSE;
ELSE
	GV.O_Steuerspannung := TRUE;
END_IF

// Variabeln Reset
GV.sys_aus := FALSE;
GV.sys_start := FALSE;
GV.sys_bereit:= FALSE;
GV.sys_betrieb := FALSE;
GV.sys_herunterfahren := FALSE;

// Execute
IF NOT GV.sys_Einschalten THEN
	ExecuteFlag := FALSE;
END_IF

// Systemzustände
CASE Systemzustand OF
	0: //Aus
	GV.sys_aus := TRUE;
	Busy := FALSE;
	GV.O_Ladeschuetz := FALSE;
	GV.O_Hauptschuetz := FALSE;
	GV.sys_MPPT_aktiv := FALSE;
	
	IF NOT ExecuteFlag AND GV.sys_Einschalten OR Auto_ein THEN
		// Entweder von Hand starten oder es wird automatisch versucht
		ExecuteFlag := TRUE;
		Busy := TRUE;
		Done := FALSE;
		IF GV.inv_ein THEN
			Systemzustand :=1;
		END_IF
	END_IF
	
	1: // Aufstarten
	GV.sys_start:= TRUE;
	GV.O_Ladeschuetz := TRUE;
	
	IF GV.r_SpannungDC > 100 THEN
		GV.O_Hauptschuetz := TRUE;
		TimerLadeschuetz(IN:= TRUE, PT:= T#2S);
	END_IF
	
	IF GV.sys_Ausschalten THEN
		Systemzustand := 0;
	END_IF
	
	IF TimerLadeschuetz.Q AND GV.inv_bereit THEN
		// Inverter ist betriebsbereit
		GV.O_Ladeschuetz := FALSE;
		Systemzustand := 2;
	END_IF
	
	2: // Bereit / Leerlauf
	GV.sys_bereit := TRUE;
	GV.sys_MPPT_aktiv := FALSE;
	IF GV.sys_Einschalten THEN
		Systemzustand := 3;
	END_IF
	
	IF GV.p_Automatik AND GV.sys_Drehzahl >= GV.p_Drehzahl_soll THEN
		Systemzustand := 3;
	END_IF
		
	IF GV.sys_Ausschalten OR GV.inv_standby THEN
		Systemzustand := 0;
	END_IF
		
	3: // Betrieb
	GV.sys_betrieb := TRUE;
	GV.sys_MPPT_aktiv := TRUE;
	
	IF GV.sys_Ausschalten THEN
		Systemzustand := 4;
	END_IF
	
	IF NOT GV.inv_betrieb AND GV.sys_Drehzahl_Sensor <= GV.p_Drehzahl_min THEN
		Systemzustand :=0;
	END_IF
	

	4: // Herunterfahren
	GV.sys_herunterfahren := TRUE;
	
	IF GV.inv_leerlauf THEN
		Systemzustand := 2;
	END_IF
END_CASE

// InfoLampe
BLINK_Starten(ENABLE := TRUE, TIMELOW := T#1S, TIMEHIGH := T#1S);
BLINK_bereit(ENABLE := TRUE, TIMELOW := T#3S, TIMEHIGH := T#3S);
BLINK_Stoerung(ENABLE := TRUE, TIMELOW := T#3S, TIMEHIGH := T#1S);
GV.O_Infolampe := 
(BLINK_Starten.OUT AND GV.sys_start OR GV.sys_herunterfahren) 
OR (GV.sys_bereit AND BLINK_bereit.OUT)
OR (GV.sammelstoerung AND BLINK_Stoerung.OUT)
OR GV.sys_betrieb;


END_IF

END_PROGRAM

// MQTTDataLogger
PROGRAM MQTTDataLogger
VAR
	fbClient     : MQTT.MQTTClient;
	
	iPublishStep : INT := 0; // 0=Start, 1=Drehzahl senden, 2=Leistung senden, 3=Warten
    fbPubDrehzahl : MQTT.MQTTPublish;
    fbPubLeistung : MQTT.MQTTPublish;

    sBrokerIP    : STRING(80) := '192.168.178.42';
    uiPort       : UINT := 1883;
    sClientID    : STRING(255) := 'SGSclient';

    xConnected   : BOOL;
    xError       : BOOL;
    sError       : STRING(255);

    // Payloads
    wsTopicDrehzahl : WSTRING(1024);
    wsTopicLeistung : WSTRING(1024);
    wsPayload       : WSTRING(255);
    sPayload        : STRING(80);

    abyPayload : ARRAY[0..255] OF BYTE;
    udiPayloadSize : UDINT;

    tLastSend  : TIME := T#0s;
    tInterval  : TIME := T#5S;
	
 // Reconnect-Logik
    xReconnectPending     : BOOL := FALSE;
    tLastError            : TIME := T#0s;
    tReconnectDelay       : TIME := T#5s;
    udiMQTTErrorCounter   : UDINT := 0;
END_VAR

// --- MQTT Client aktivieren ---
xConnected := fbClient.xConnectedToBroker;
xError := fbClient.xError;

// Standard: Verbindung aktiv halten
fbClient.xEnable := TRUE;

IF xError THEN
    sError := CONCAT('MQTT Fehler: ', TO_STRING(fbClient.eMQTTError));

    // Reconnect auslösen nach Delay
    IF (TIME() - tLastError) >= tReconnectDelay THEN
        fbClient.xEnable := FALSE;
        xReconnectPending := TRUE;
        tLastError := TIME();
        udiMQTTErrorCounter := udiMQTTErrorCounter + 1;
    END_IF;

    IF udiMQTTErrorCounter >= 100 THEN
        GV.stoerung_MQTT := TRUE;
    END_IF
ELSE
    sError := '';
    xReconnectPending := FALSE;
    udiMQTTErrorCounter := 0;
    GV.stoerung_MQTT := FALSE;
END_IF

// Reconnect aktivieren nach Trennung
IF xReconnectPending AND (TIME() - tLastError >= T#1s) THEN
    fbClient.xEnable := TRUE;
END_IF

// --- MQTT Client aufrufen ---
fbClient(
    xEnable := fbClient.xEnable,
    sHostname := sBrokerIP,
    uiPort := uiPort,
    sClientId := sClientID
);

// --- Nur senden wenn verbunden und Intervall erreicht ---
IF xConnected AND (TIME() - tLastSend >= tInterval) THEN
    CASE iPublishStep OF

        0: // Init Drehzahl
            sPayload := REAL_TO_STRING(GV.sys_Drehzahl);
            wsPayload := TO_WSTRING(sPayload);
            wsTopicDrehzahl := TO_WSTRING('SGS/Drehzahl');
            udiPayloadSize := WSTRING_TO_BYTEARRAY_UTF8(wsPayload, ADR(abyPayload), SIZEOF(abyPayload));
            iPublishStep := 1;

        1: // Publish Drehzahl
            IF NOT fbPubDrehzahl.xBusy AND NOT fbPubDrehzahl.xDone THEN
                fbPubDrehzahl.xExecute := TRUE;
            ELSE
                fbPubDrehzahl.xExecute := FALSE;
            END_IF;

            fbPubDrehzahl(
                xExecute := fbPubDrehzahl.xExecute,
                mqttClient := fbClient,
                wsTopicName := wsTopicDrehzahl,
                eQoS := MQTT.MQTT_QOS.QoS0,
                xRetain := FALSE,
                xReDelivery := FALSE,
                pbPayload := ADR(abyPayload),
                udiPayloadSize := udiPayloadSize
            );

            IF fbPubDrehzahl.xDone THEN
                iPublishStep := 2;
            END_IF;

        2: // Init Leistung
            sPayload := REAL_TO_STRING(GV.r_LeistungAC);
            wsPayload := TO_WSTRING(sPayload);
            wsTopicLeistung := TO_WSTRING('SGS/Leistung');
            udiPayloadSize := WSTRING_TO_BYTEARRAY_UTF8(wsPayload, ADR(abyPayload), SIZEOF(abyPayload));
            iPublishStep := 3;

        3: // Publish Leistung
            IF NOT fbPubLeistung.xBusy AND NOT fbPubLeistung.xDone THEN
                fbPubLeistung.xExecute := TRUE;
            ELSE
                fbPubLeistung.xExecute := FALSE;
            END_IF;

            fbPubLeistung(
                xExecute := fbPubLeistung.xExecute,
                mqttClient := fbClient,
                wsTopicName := wsTopicLeistung,
                eQoS := MQTT.MQTT_QOS.QoS0,
                xRetain := FALSE,
                xReDelivery := FALSE,
                pbPayload := ADR(abyPayload),
                udiPayloadSize := udiPayloadSize
            );

            IF fbPubLeistung.xDone THEN
                tLastSend := TIME();      // Zeitstempel setzen
                iPublishStep := 0;        // Wieder von vorne
            END_IF;
    END_CASE;
END_IF

END_PROGRAM

// PLC_AC500_V3/Application/PLC_PRG
PROGRAM PLC_PRG
VAR
	Systemzustand: INT;
	Busy: BOOL;
	
	ExecuteFlag: BOOL;
	Done: BOOL;
	TimerLadeschuetz :TON;
	
	
	BLINK_Starten: BLINK;
	BLINK_bereit: BLINK;
	BLINK_Stoerung: BLINK;
END_VAR

// Bedienknöpfe

GV.sys_Einschalten := GV.I_Einschalten OR GV.v_Einschalten;
GV.sys_Ausschalten := GV.I_Ausschalten OR GV.v_Ausschalten;

// Störung überprüfen
IF GV.sammelstoerung THEN
	GV.O_Steuerspannung := FALSE;
	Systemzustand := 0;
	
ELSE
// Störungsfrei, Steuerspannung freigeben	

IF NOT GV.inv_ein THEN
		Systemzustand := 0;
END_IF
	
IF GV.I_Notaus THEN
	GV.O_Steuerspannung:= FALSE;
ELSE
	GV.O_Steuerspannung := TRUE;
END_IF

// Variabeln Reset
GV.sys_aus := FALSE;
GV.sys_start := FALSE;
GV.sys_bereit:= FALSE;
GV.sys_betrieb := FALSE;
GV.sys_herunterfahren := FALSE;

// Execute
IF NOT GV.sys_Einschalten THEN
	ExecuteFlag := FALSE;
END_IF

// Systemzustände
CASE Systemzustand OF
	0: //Aus
	GV.sys_aus := TRUE;
	Busy := FALSE;
	GV.O_Ladeschuetz := FALSE;
	GV.O_Hauptschuetz := FALSE;
	GV.sys_MPPT_aktiv := FALSE;
	
	IF GV.sys_Einschalten AND NOT ExecuteFlag THEN
		ExecuteFlag := TRUE;
		Busy := TRUE;
		Done := FALSE;
		IF GV.inv_ein THEN
			Systemzustand :=1;
		END_IF
	END_IF
	
	1: // Aufstarten
	GV.sys_start:= TRUE;
	GV.O_Ladeschuetz := TRUE;
	
	IF GV.r_SpannungDC > 100 THEN
		GV.O_Hauptschuetz := TRUE;
		TimerLadeschuetz(IN:= TRUE, PT:= T#2S);
	END_IF
	
	IF GV.sys_Ausschalten THEN
		Systemzustand := 0;
	END_IF
	
	IF TimerLadeschuetz.Q AND GV.inv_bereit THEN
		GV.O_Ladeschuetz := FALSE;
		Systemzustand := 2;
	END_IF
	
	2: // Bereit
	GV.sys_bereit := TRUE;
	GV.sys_MPPT_aktiv := FALSE;
	IF GV.sys_Einschalten THEN
		Systemzustand := 3;
	END_IF
		
	IF GV.sys_Ausschalten THEN
		Systemzustand := 0;
	END_IF
		
	3: // Betrieb
	GV.sys_betrieb := TRUE;
	GV.sys_MPPT_aktiv := TRUE;
	
	IF GV.sys_Ausschalten THEN
		Systemzustand := 4;
	END_IF
	
	4: // Herunterfahren
	GV.sys_herunterfahren := TRUE;
	
	IF GV.inv_leerlauf THEN
		Systemzustand := 2;
	END_IF
END_CASE

// InfoLampe
BLINK_Starten(ENABLE := TRUE, TIMELOW := T#1S, TIMEHIGH := T#1S);
BLINK_bereit(ENABLE := TRUE, TIMELOW := T#3S, TIMEHIGH := T#3S);
BLINK_Stoerung(ENABLE := TRUE, TIMELOW := T#3S, TIMEHIGH := T#1S);
GV.O_Infolampe := 
(GV.sys_start OR GV.sys_herunterfahren AND BLINK_Starten.OUT) 
OR (GV.sys_bereit AND BLINK_bereit.OUT)
OR (GV.sammelstoerung AND BLINK_Stoerung.OUT)
OR GV.sys_betrieb;


END_IF

END_PROGRAM

// Schaltlogik
PROGRAM Schaltlogik
VAR
	
Ladeschuetz_ein		:BOOL :=FALSE;
	RS_Einschalten: RS;
	RS_Hauptschuetz_Freigabe: RS;
	RS_Hauptschuetz: RS;
	TON_Laden_delay: TON;
	RS_Ladeschuetz: RS;
	TP_Ladeschuetz: TP;
	TP_Steuerspannung: TP;
	RS_Steuerspannung: RS;
	TP_Hauptschuetz: TP;
	RS_Ausschalten: RS;
	RS_Inverter_start: RS;
	TP_Inverter_start: TP;
	RS_sys_start: RS;
	TON_Einschaltverzoegerung: TON;
	RS_sys_Betrieb: RS;
	TP_sys_betrieb: TP;
	TP_sys_start: TP;
	RS_sys_aus: RS;
	TP_Sys_aus: TP;
	RS_bereit: RS;
	TP_Visu_ein: TP;
	TP_Visu_aus: TP;
	OBIOForwardCounter_0: OBIOForwardCounter;

	TP_Einschalten: TP;
	RS_sys_bereit: RS;
	TP_sys_bereit: TP;
	TP_aufstarten: TP;
	TON_sys_aus: TON;
	TON_Hauptschuetz: TON;
	TON_Ladeschuetz: TON;
	BLINK_Infolampe: BLINK;
	BLINK_Starten: BLINK;
	BLINK_bereit: BLINK;
	BLINK_Stoerung: BLINK;
	TON_system_aus: TON;
END_VAR

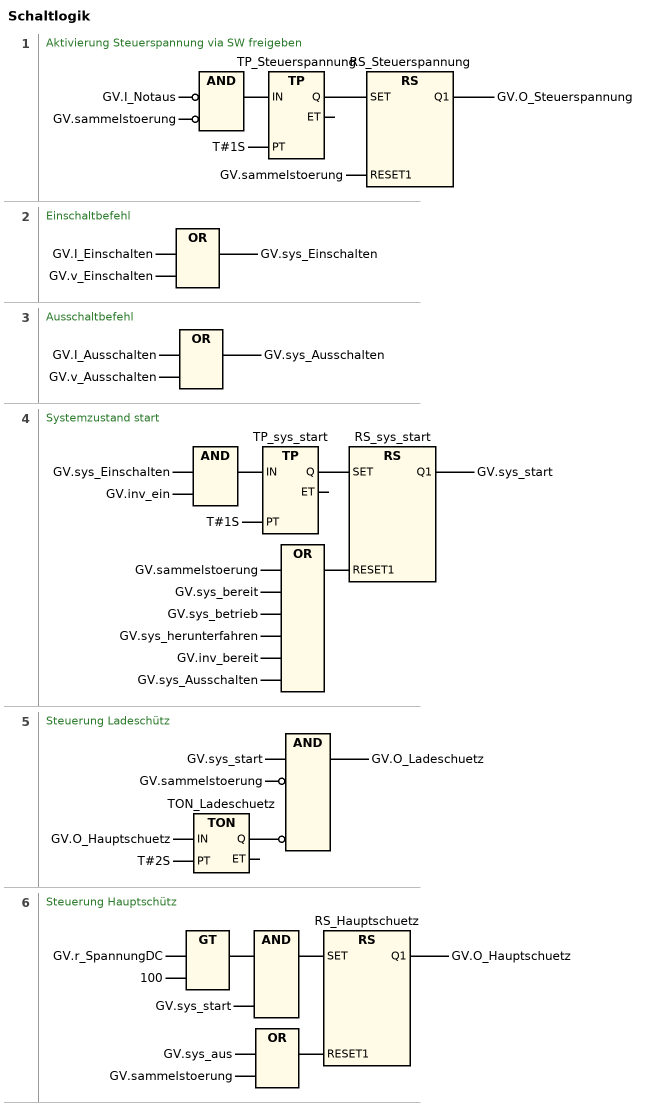
// NETWORK 1
// Aktivierung Steuerspannung via SW freigeben
TP_Steuerspannung(IN := NOT GV.I_Notaus AND NOT GV.sammelstoerung, PT := T#1S); // TP
RS_Steuerspannung(SET := TP_Steuerspannung.Q, RESET1 := GV.sammelstoerung); // RS
GV.O_Steuerspannung := RS_Steuerspannung.Q1;

// NETWORK 2
// Einschaltbefehl
GV.sys_Einschalten := GV.I_Einschalten OR GV.v_Einschalten;

// NETWORK 3
// Ausschaltbefehl
GV.sys_Ausschalten := GV.I_Ausschalten OR GV.v_Ausschalten;

// NETWORK 4
// Systemzustand start
TP_sys_start(IN := GV.sys_Einschalten AND GV.inv_ein, PT := T#1S); // TP
RS_sys_start(SET := TP_sys_start.Q, RESET1 := GV.sammelstoerung OR GV.sys_bereit OR GV.sys_betrieb OR GV.sys_herunterfahren OR GV.inv_bereit OR GV.sys_Ausschalten); // RS
GV.sys_start := RS_sys_start.Q1;

// NETWORK 5
// Steuerung Ladeschütz
TON_Ladeschuetz(IN := GV.O_Hauptschuetz, PT := T#2S); // TON
GV.O_Ladeschuetz := GV.sys_start AND NOT GV.sammelstoerung AND NOT TON_Ladeschuetz.Q;

// NETWORK 6
// Steuerung Hauptschütz
RS_Hauptschuetz(SET := GV.r_SpannungDC > 100 AND GV.sys_start, RESET1 := GV.sys_aus OR GV.sammelstoerung); // RS
GV.O_Hauptschuetz := RS_Hauptschuetz.Q1;

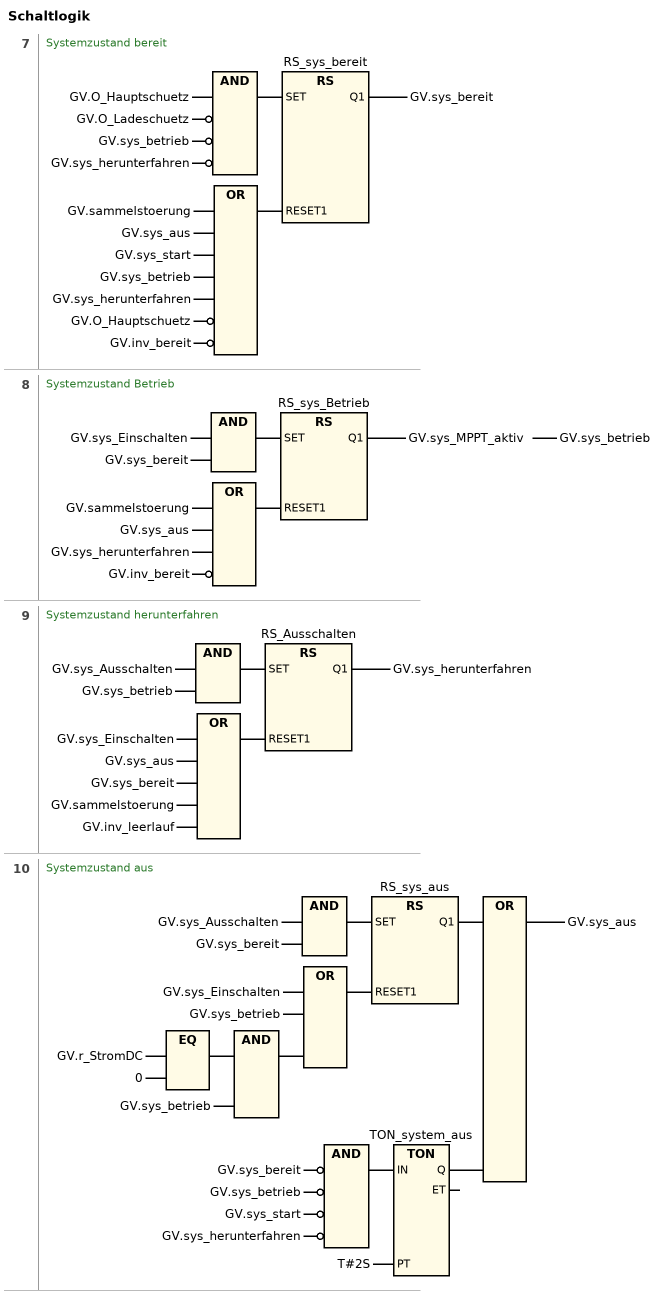
// NETWORK 7
// Systemzustand bereit
RS_sys_bereit(SET := GV.O_Hauptschuetz AND NOT GV.O_Ladeschuetz AND NOT GV.sys_betrieb AND NOT GV.sys_herunterfahren, RESET1 := GV.sammelstoerung OR GV.sys_aus OR GV.sys_start OR GV.sys_betrieb OR GV.sys_herunterfahren OR NOT GV.O_Hauptschuetz OR NOT GV.inv_bereit); // RS
GV.sys_bereit := RS_sys_bereit.Q1;

// NETWORK 8
// Systemzustand Betrieb
RS_sys_Betrieb(SET := GV.sys_Einschalten AND GV.sys_bereit, RESET1 := GV.sammelstoerung OR GV.sys_aus OR GV.sys_herunterfahren OR NOT GV.inv_bereit); // RS
GV.sys_MPPT_aktiv := RS_sys_Betrieb.Q1;
GV.sys_betrieb := RS_sys_Betrieb.Q1;

// NETWORK 9
// Systemzustand herunterfahren
RS_Ausschalten(SET := GV.sys_Ausschalten AND GV.sys_betrieb, RESET1 := GV.sys_Einschalten OR GV.sys_aus OR GV.sys_bereit OR GV.sammelstoerung OR GV.inv_leerlauf); // RS
GV.sys_herunterfahren := RS_Ausschalten.Q1;

// NETWORK 10
// Systemzustand aus
RS_sys_aus(SET := GV.sys_Ausschalten AND GV.sys_bereit, RESET1 := GV.sys_Einschalten OR GV.sys_betrieb OR GV.r_StromDC = 0 AND GV.sys_betrieb); // RS
TON_system_aus(IN := NOT GV.sys_bereit AND NOT GV.sys_betrieb AND NOT GV.sys_start AND NOT GV.sys_herunterfahren, PT := T#2S); // TON
GV.sys_aus := RS_sys_aus.Q1 OR TON_system_aus.Q;

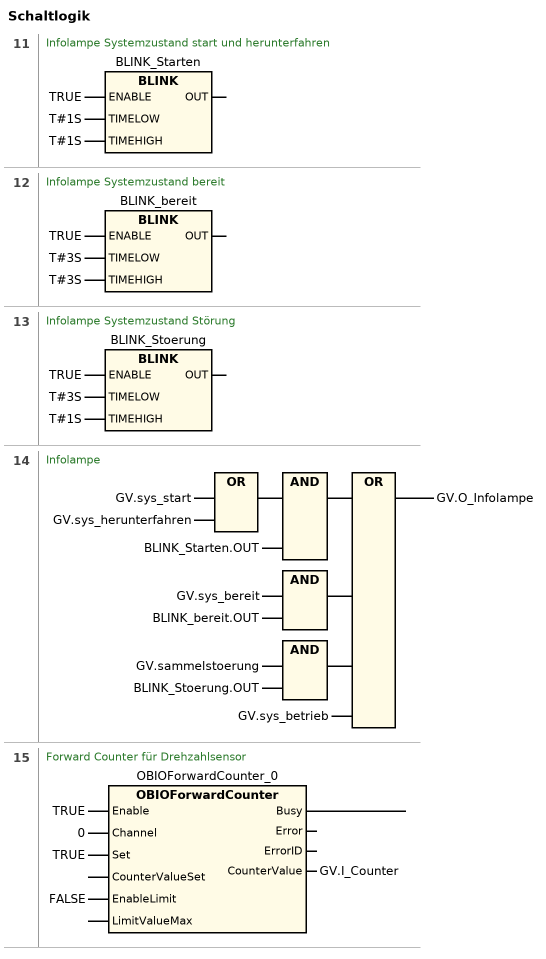
// NETWORK 11
// Infolampe Systemzustand start und herunterfahren
BLINK_Starten(ENABLE := TRUE, TIMELOW := T#1S, TIMEHIGH := T#1S); // BLINK

// NETWORK 12
// Infolampe Systemzustand bereit
BLINK_bereit(ENABLE := TRUE, TIMELOW := T#3S, TIMEHIGH := T#3S); // BLINK

// NETWORK 13
// Infolampe Systemzustand Störung
BLINK_Stoerung(ENABLE := TRUE, TIMELOW := T#3S, TIMEHIGH := T#1S); // BLINK

// NETWORK 14
// Infolampe
GV.O_Infolampe := (GV.sys_start OR GV.sys_herunterfahren) AND BLINK_Starten.OUT OR GV.sys_bereit AND BLINK_bereit.OUT OR GV.sammelstoerung AND BLINK_Stoerung.OUT OR GV.sys_betrieb;

// NETWORK 15
// Forward Counter für Drehzahlsensor
OBIOForwardCounter_0(
    Enable := TRUE,
    Channel := 0,
    Set := TRUE,
    EnableLimit := FALSE,
    CounterValue => GV.I_Counter); // OBIOForwardCounter

END_PROGRAM

// WSTRING_Concat
FUNCTION WSTRING_Concat : WSTRING(512)
VAR_INPUT
    ws1 : WSTRING(512);
    ws2 : WSTRING(512);
END_VAR
VAR
    len1 : INT;
    len2 : INT;
    i : INT;
END_VAR


    // Länge ws1 bestimmen (bis Null-Terminator)
    len1 := 0;
    WHILE (len1 < 512) AND (ws1[len1 + 1] <> 0) DO
        len1 := len1 + 1;
    END_WHILE;

    // Länge ws2 bestimmen
    len2 := 0;
    WHILE (len2 < 512) AND (ws2[len2 + 1] <> 0) DO
        len2 := len2 + 1;
    END_WHILE;

    // ws1 in Ergebnis kopieren
    FOR i := 1 TO len1 DO
        WSTRING_Concat[i] := ws1[i];
    END_FOR

    // ws2 anhängen, aber nicht über max Länge hinaus
    FOR i := 1 TO len2 DO
        IF (len1 + i) <= 512 THEN
            WSTRING_Concat[len1 + i] := ws2[i];
        ELSE
            EXIT;
        END_IF
    END_FOR

    // Null-Terminator anfügen
    IF (len1 + len2 + 1) <= 512 THEN
        WSTRING_Concat[len1 + len2 + 1] := 0;
    END_IF

END_FUNCTION

// Visualisierung/Uebersicht
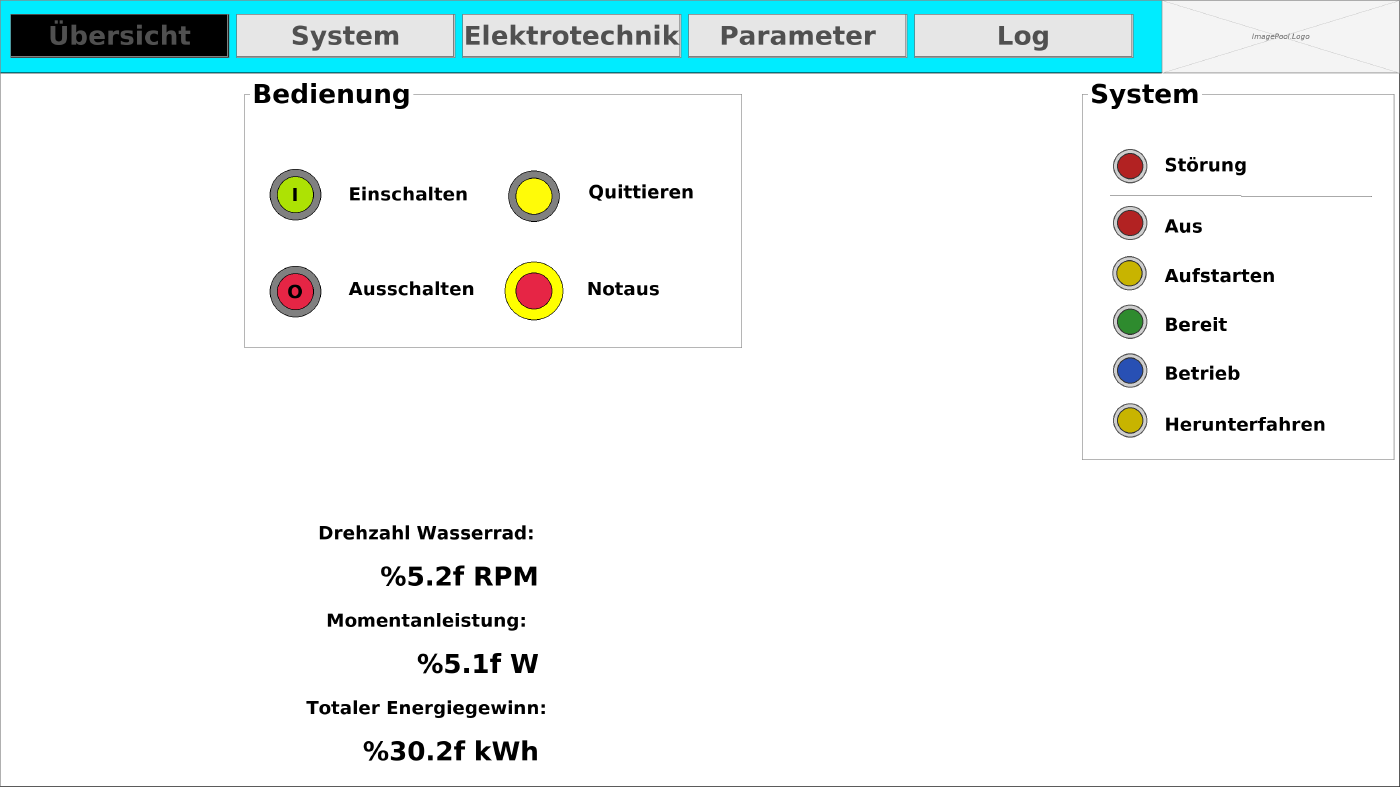
VISUALIZATION Uebersicht  // 1920x1080
    Rectangle (0,0 1920x1080)
    GroupBox (1484,121 428x510), "System"
        Lamp1 (39,426 54x60), variable: GV.sys_herunterfahren, style: Lamp-Lamp1-Yellow
        Label (110,436 218x50), "Herunterfahren"
        Lamp1 (39,359 54x57), variable: GV.sys_betrieb, style: Lamp-Lamp1-Blue
        Label (110,366 200x50), "Betrieb"
        Lamp1 (39,158 54x54), variable: GV.sys_aus, style: Lamp-Lamp1-Red
        Lamp1 (38,224 54x60), variable: GV.sys_start, style: Lamp-Lamp1-Yellow
        Label (110,164 200x50), "Aus"
        Label (110,232 200x50), "Aufstarten"
        Label (110,299 200x50), "Bereit"
        Lamp1 (39,292 54x57), variable: GV.sys_bereit, style: Lamp-Lamp1-Green
        Lamp1 (39,80 54x54), variable: GV.sammelstoerung, style: Lamp-Lamp1-Red
        Label (110,80 225x50), "Störung"
        Line (39,147) (397,148)
    Rectangle (268,1006 474x50), "%30.2f kWh", text variable: GV.r_Energie
    Rectangle (450,766 292x50), "%5.2f RPM", text variable: GV.sys_Drehzahl_Wasserrad
    Rectangle (496,886 246x50), "%5.1f W", text variable: GV.r_LeistungAC
    GroupBox (335,121 682x356), "Bedienung"
        Rectangle (140,120 250x50), "Einschalten"
        Rectangle (140,250 250x50), "Ausschalten"
        Ellipse (35,111 70x70)
        Ellipse (45,121 50x50), "I"
            tap GV.v_Einschalten
        Ellipse (35,244 70x70)
        Ellipse (45,254 50x50), "O"
            tap GV.v_Ausschalten
        Ellipse (362,113 70x70)
        Ellipse (372,123 50x50)
            tap GV.stoerung_quittieren
        Rectangle (467,250 200x50), "Notaus"
    Ellipse (692,359 80x80)
    Ellipse (707,374 50x50)
        tap GV.v_Notaus
    Label (428,706 314x50), "Drehzahl Wasserrad:"
    Rectangle (804,238 200x50), "Quittieren"
    Label (428,826 314x50), "Momentanleistung:"
    Label (428,946 314x50), "Totaler Energiegewinn:"
    Rectangle (1555,891 150x30)
    Rectangle (0,0 1920x100)
    Button (944,19 300x60), "Parameter"
        OnMouseClick:  Assign=Parameter, Type=Assignment
    Button (324,19 300x60), "System"
        OnMouseClick:  Assign=System, Type=Assignment
    Button (634,19 300x60), "Elektrotechnik"
        OnMouseClick:  Assign=Elektrotechnik, Type=Assignment
    Button (14,19 300x60), "Übersicht"
        OnMouseClick:  Assign=Uebersicht, Type=Assignment
    Button (1254,19 300x60), "Log"
        OnMouseClick:  Assign=Logging, Type=Assignment
    Image (1593,0 327x100), image: ImagePool.Logo
        OnMouseClick:  Assign=Show, Type=Assignment
END_VISUALIZATION

// Visualisierung/Elektrotechnik
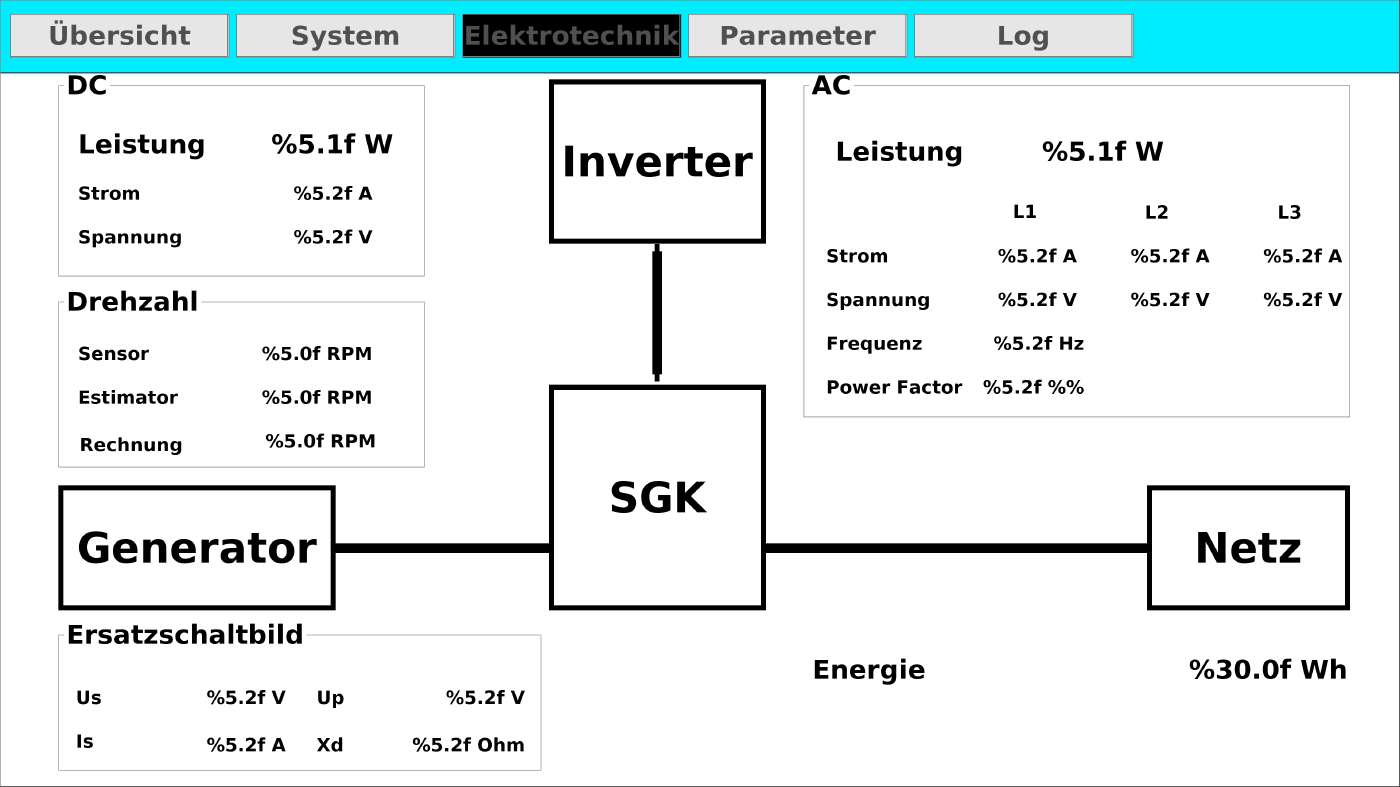
VISUALIZATION Elektrotechnik  // 1920x1080
    Rectangle (0,0 1920x1080)
    Rectangle (409,749 370x6)
        toggle GV.v_Geni_lauft
    RoundedRectangle (753,109 297x225), "Inverter"
    RoundedRectangle (80,666 380x171), "Generator"
    Rectangle (1018,749 581x6)
        toggle GV.sys_betrieb
    RoundedRectangle (753,528 297x309), "SGK"
    Rectangle (807,426 188x6), angle 90
        toggle GV.sys_betrieb
    GroupBox (1102,109 749x463), "AC"
        Rectangle (410,157 150x50), "L2"
        Rectangle (592,157 150x50), "L3"
        Rectangle (238,337 150x50), "%5.2f Hz", text variable: GV.r_Frequenz
        Rectangle (28,337 200x50), "Frequenz"
        Rectangle (28,397 200x50), "Power Factor"
        Rectangle (238,397 150x50), "%5.2f %%", text variable: GV.r_PF
        Rectangle (592,277 150x50), "%5.2f V", text variable: GV.r_StrangspannungC
        Rectangle (410,277 150x50), "%5.2f V", text variable: GV.r_StrangspannungB
        Rectangle (228,277 150x50), "%5.2f V", text variable: GV.r_StrangspannungA
        Rectangle (592,217 150x50), "%5.2f A", text variable: GV.r_StromPhaseB
        Rectangle (410,217 150x50), "%5.2f A", text variable: GV.r_StromPhaseB
        Rectangle (28,277 200x50), "Spannung"
        Rectangle (28,217 200x50), "Strom"
        Rectangle (228,217 150x50), "%5.2f A", text variable: GV.r_StromPhaseA
        Rectangle (229,156 150x50), "L1"
        Rectangle (251,74 246x50), "%5.1f W", text variable: GV.r_LeistungAC
        Rectangle (41,74 200x50), "Leistung"
    Rectangle (1321,894 530x50), "%30.0f Wh", text variable: GV.r_EnergieDC
    Rectangle (1111,894 200x50), "Energie"
    GroupBox (80,109 502x270), "DC"
        Rectangle (24,131 200x50), "Strom"
        Rectangle (24,191 200x50), "Spannung"
        Rectangle (234,131 200x50), "%5.2f A", text variable: GV.r_StromDC
        Rectangle (234,191 200x50), "%5.2f V", text variable: GV.r_SpannungDC
        Rectangle (24,64 200x50), "Leistung"
        Rectangle (234,64 228x50), "%5.1f W", text variable: GV.r_LeistungDC
    RoundedRectangle (1573,666 278x171), "Netz"
    GroupBox (80,406 502x235), "Drehzahl"
        Rectangle (24,54 200x50), "Sensor"
        Rectangle (24,114 200x50), "Estimator"
        Rectangle (234,54 200x50), "%5.0f RPM", text variable: GV.sys_Drehzahl_Sensor
        Rectangle (234,114 200x50), "%5.0f RPM", text variable: GV.sys_Drehzahl_Estimator
        Rectangle (26,179 200x50), "Rechnung"
        Rectangle (239,174 200x50), "%5.0f RPM", text variable: GV.sys_Drehzahl_Rechner
    GroupBox (80,863 662x194), "Ersatzschaltbild"
        Rectangle (443,69 200x50), "%5.2f V", text variable: Berechnungen.U_p
        Rectangle (351,69 80x50), "Up"
        Rectangle (115,134 200x50), "%5.2f A", text variable: Berechnungen.I_s
        Rectangle (115,69 200x50), "%5.2f V", text variable: Berechnungen.U_s
        Rectangle (21,129 80x50), "Is"
        Rectangle (21,69 80x50), "Us"
        Rectangle (443,134 200x50), "%5.2f Ohm", text variable: Berechnungen.X_d
        Rectangle (351,134 80x50), "Xd"
    Rectangle (0,0 1920x100)
    Button (944,19 300x60), "Parameter"
        OnMouseClick:  Assign=Parameter, Type=Assignment
    Button (324,19 300x60), "System"
        OnMouseClick:  Assign=System, Type=Assignment
    Button (634,19 300x60), "Elektrotechnik"
        OnMouseClick:  Assign=Elektrotechnik, Type=Assignment
    Button (14,19 300x60), "Übersicht"
        OnMouseClick:  Assign=Uebersicht, Type=Assignment
    Button (1254,19 300x60), "Log"
        OnMouseClick:  Assign=Logging, Type=Assignment
END_VISUALIZATION

// Visualisierung/System
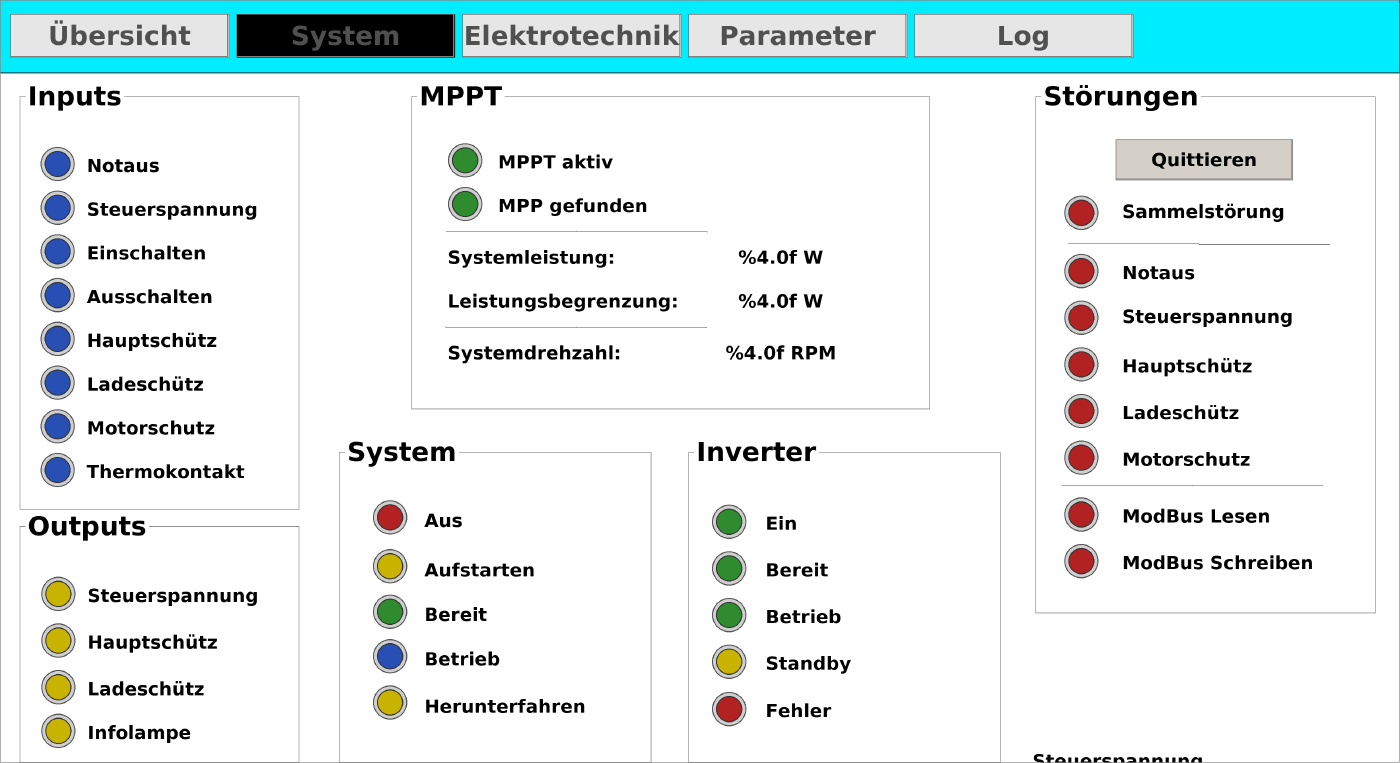
VISUALIZATION System  // 1920x1047
    GroupBox (465,612 428x435), "System"
        Label (948,407 250x50), "Steuerspannung"
        Lamp1 (43,199 54x57), variable: GV.sys_bereit, style: Lamp-Lamp1-Green
        Label (114,206 200x50), "Bereit"
        Label (114,145 200x50), "Aufstarten"
        Label (114,77 200x50), "Aus"
        Lamp1 (43,135 54x60), variable: GV.sys_start, style: Lamp-Lamp1-Yellow
        Lamp1 (43,71 54x54), variable: GV.sys_aus, style: Lamp-Lamp1-Red
        Label (114,267 200x50), "Betrieb"
        Lamp1 (43,260 54x57), variable: GV.sys_betrieb, style: Lamp-Lamp1-Blue
        Label (114,332 218x50), "Herunterfahren"
        Lamp1 (43,322 54x60), variable: GV.sys_herunterfahren, style: Lamp-Lamp1-Yellow
    GroupBox (1420,124 466x717), "Störungen"
        Button (110,67 243x56), "Quittieren"
            tap GV.stoerung_quittieren
        Lamp1 (36,619 54x54), variable: GV.stoerung_Modbus_Schreiben, style: Lamp-Lamp1-Red
    GroupBox (27,714 383x333), "Outputs"
        Label (90,78 250x50), "Steuerspannung"
        Label (90,206 250x50), "Ladeschütz"
        Label (90,142 250x50), "Hauptschütz"
        Lamp1 (26,202 54x54), variable: GV.O_Ladeschuetz, style: Lamp-Lamp1-Yellow
        Lamp1 (26,138 54x54), variable: GV.O_Hauptschuetz, style: Lamp-Lamp1-Yellow
        Lamp1 (26,74 54x54), variable: GV.O_Steuerspannung, style: Lamp-Lamp1-Yellow
        Label (90,266 250x50), "Infolampe"
        Lamp1 (26,262 54x54), variable: GV.O_Infolampe, style: Lamp-Lamp1-Yellow
    Line (1456,665) (1814,666)
    Lamp1 (1456,345 54x54), variable: GV.stoerung_Notaus, style: Lamp-Lamp1-Red
    Label (1536,349 350x50), "Notaus"
    Lamp1 (1456,409 54x54), variable: GV.stoerung_Steuerspannung, style: Lamp-Lamp1-Red
    Label (1536,409 350x50), "Steuerspannung"
    Lamp1 (1456,473 54x54), variable: GV.stoerung_Hauptschuetz, style: Lamp-Lamp1-Red
    Label (1536,477 350x50), "Hauptschütz"
    Lamp1 (1456,537 54x54), variable: GV.stoerung_Ladeschuetz, style: Lamp-Lamp1-Red
    Label (1536,541 350x50), "Ladeschütz"
    Lamp1 (1456,601 54x54), variable: GV.stoerung_Motorschutz, style: Lamp-Lamp1-Red
    Label (1536,605 350x50), "Motorschutz"
    Lamp1 (1456,265 54x54), variable: GV.sammelstoerung, style: Lamp-Lamp1-Red
    Label (1536,265 350x50), "Sammelstörung"
    Line (1465,334) (1823,335)
    Lamp1 (1456,679 54x54), variable: GV.stoerung_Modbus_Lesen, style: Lamp-Lamp1-Red
    Label (1536,747 350x50), "ModBus Schreiben"
    Label (1536,683 350x50), "ModBus Lesen"
    GroupBox (944,612 428x435), "Inverter"
        Lamp1 (29,334 54x54), variable: GV.inv_fehler, style: Lamp-Lamp1-Red
        Label (103,338 217x50), "Fehler"
        Lamp1 (29,269 54x54), variable: GV.inv_standby, style: Lamp-Lamp1-Yellow
        Label (103,273 217x50), "Standby"
        Lamp1 (29,205 54x54), variable: GV.inv_betrieb, style: Lamp-Lamp1-Green
        Label (103,209 217x50), "Betrieb"
        Lamp1 (29,141 54x54), variable: GV.inv_bereit, style: Lamp-Lamp1-Green
        Label (103,145 217x50), "Bereit"
        Lamp1 (29,77 54x54), variable: GV.inv_ein, style: Lamp-Lamp1-Green
        Label (103,81 217x50), "Ein"
    GroupBox (27,124 383x575), "Inputs"
        Label (89,78 250x50), "Notaus"
        Lamp1 (25,74 54x54), variable: GV.I_Notaus, style: Lamp-Lamp1-Blue
        Label (89,138 250x50), "Steuerspannung"
        Lamp1 (25,134 54x54), variable: GV.I_Steuerspannung, style: Lamp-Lamp1-Blue
        Label (89,198 250x50), "Einschalten"
        Lamp1 (25,194 54x54), variable: GV.sys_Einschalten, style: Lamp-Lamp1-Blue
        Label (89,258 250x50), "Ausschalten"
        Lamp1 (25,254 54x54), variable: GV.sys_Ausschalten, style: Lamp-Lamp1-Blue
        Label (89,318 250x50), "Hauptschütz"
        Lamp1 (25,314 54x54), variable: GV.I_Hauptschuetz, style: Lamp-Lamp1-Blue
        Label (89,378 250x50), "Ladeschütz"
        Lamp1 (25,374 54x54), variable: GV.I_Ladeschuetz, style: Lamp-Lamp1-Blue
        Label (89,438 250x50), "Motorschutz"
        Lamp1 (25,434 54x54), variable: GV.I_Motorschutz, style: Lamp-Lamp1-Blue
        Label (89,498 250x50), "Thermokontakt"
        Lamp1 (25,494 54x54), variable: GV.I_Temperatur, style: Lamp-Lamp1-Blue
    GroupBox (564,124 711x437), "MPPT"
        Label (47,204 350x50), "Systemleistung:"
        Line (48,193) (406,194)
        Textfield (407,204 200x50), "%4.0f W", text variable: GV.r_LeistungAC
        Label (47,264 350x50), "Leistungsbegrenzung:"
        Textfield (407,264 200x50), "%4.0f W", text variable: Inverter.zielLeistung
        Label (116,73 217x50), "MPPT aktiv"
        Lamp1 (47,69 54x54), variable: GV.sys_MPPT_aktiv, style: Lamp-Lamp1-Green
        Label (116,133 217x50), "MPP gefunden"
        Lamp1 (47,129 54x54), variable: GV.sys_MPP_erreicht, style: Lamp-Lamp1-Green
        Line (47,324) (405,325)
        Label (47,335 350x50), "Systemdrehzahl:"
        Textfield (407,335 200x50), "%4.0f RPM", text variable: GV.sys_Drehzahl
    Rectangle (0,0 1920x100)
    Button (944,19 300x60), "Parameter"
        OnMouseClick:  Assign=Parameter, Type=Assignment
    Button (324,19 300x60), "System"
        OnMouseClick:  Assign=System, Type=Assignment
    Button (634,19 300x60), "Elektrotechnik"
        OnMouseClick:  Assign=Elektrotechnik, Type=Assignment
    Button (14,19 300x60), "Übersicht"
        OnMouseClick:  Assign=Uebersicht, Type=Assignment
    Button (1254,19 300x60), "Log"
        OnMouseClick:  Assign=Logging, Type=Assignment
END_VISUALIZATION

// Visualisierung/Parameter
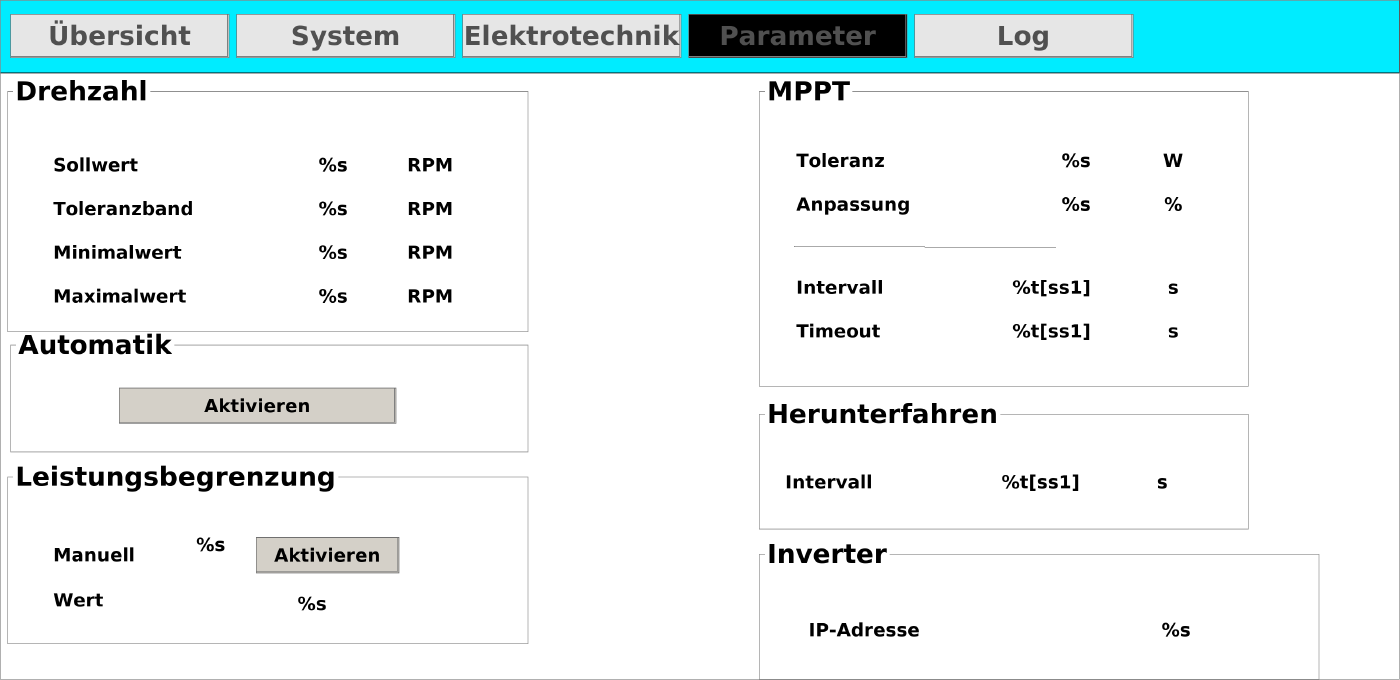
VISUALIZATION Parameter  // 1920x933
    GroupBox (1041,117 671x413), "MPPT"
        Line (48,221) (406,222)
        Label (48,78 250x50), "Toleranz"
        Textfield (308,78 150x50), "%s", tooltip "Differenz zwischen eingestellter und effektiver Leistung des Inverters, sodass es als "erreicht" gilt.", text variable: GV.p_Leistung_Toleranz
            OnMouseClick: write the text variable via VisuDialogs.Numpad
        Textfield (518,78 100x50), "W"
            OnMouseClick: write the text variable via Edit
        Label (48,138 250x50), "Anpassung"
        Textfield (308,138 150x50), "%s", tooltip "Leistungsanpassungsschritt, die pro Intervall gemacht wird. Input von 10 bedeutet 0.1%", text variable: GV.p_Leistung_Anpassung
            OnMouseClick: write the text variable via VisuDialogs.Keypad, min 0, max 5000
        Textfield (518,138 100x50), "%"
            OnMouseClick: write the text variable via Edit
        Label (48,252 250x50), "Intervall"
        Textfield (308,252 150x50), "%t[ss1]", tooltip "Wie lange zwischen zwei Anpassungsschritten gewartet wird.", text variable: GV.p_MPPT_Intervall
            OnMouseClick: write the text variable via VisuDialogs.Numpad
        Textfield (518,252 100x50), "s"
            OnMouseClick: write the text variable via Edit
        Label (48,312 250x50), "Timeout"
        Textfield (308,312 150x50), "%t[ss1]", tooltip "Wie lange gewartet wird, bis die Leistung als "nicht erreicht" gilt.", text variable: GV.p_MPPT_Timeout
            OnMouseClick: write the text variable via VisuDialogs.Numpad
        Textfield (518,312 100x50), "s"
            OnMouseClick: write the text variable via Edit
        Textfield (-879,605 150x50), "%s", tooltip "Manuell gesetzte Leistungsbegrenzung des Inverters, Input von 2500 resultiert in 25.00% von Pmax", text variable: GV.v_LeistungBegrenzung
            OnMouseClick: write the text variable via VisuDialogs.Numpad
    GroupBox (10,117 714x338), "Drehzahl"
        Label (60,84 250x50), "Sollwert"
        Textfield (320,84 150x50), "%s", tooltip "Sollwert der Drehzahl in RPM", text variable: GV.p_Drehzahl_soll
            OnMouseClick: write the text variable via VisuDialogs.Numpad
        Textfield (530,84 100x50), "RPM"
            OnMouseClick: write the text variable via Edit
        Label (60,144 250x50), "Toleranzband"
        Textfield (320,144 150x50), "%s", tooltip "Genauigkeit der Drehzahlregulierung. Achtung, ist der Anpassungsschritt zu gross, pendelt der MPPT", text variable: GV.p_Drehzahl_Toleranz
            OnMouseClick: write the text variable via VisuDialogs.Numpad
        Textfield (530,144 100x50), "RPM"
            OnMouseClick: write the text variable via Edit
        Label (60,204 250x50), "Minimalwert"
        Textfield (320,204 150x50), "%s", tooltip "Minimale Drehzahl. Ist die Systemdrehzahl darunter schaltet das System ab.", text variable: GV.p_Drehzahl_min
            OnMouseClick: write the text variable via VisuDialogs.Numpad
        Textfield (530,204 100x50), "RPM"
            OnMouseClick: write the text variable via Edit
        Label (60,264 250x50), "Maximalwert"
        Textfield (320,264 150x50), "%s", tooltip "Maximale Drehzahl. Ist die Systemdrehzahl darüber schaltet das System ab.", text variable: GV.p_Drehzahl_max
            OnMouseClick: write the text variable via VisuDialogs.Numpad
        Textfield (530,264 100x50), "RPM"
            OnMouseClick: write the text variable via Edit
    GroupBox (1041,560 671x166), "Herunterfahren"
        Label (33,76 250x50), "Intervall"
        Textfield (293,76 150x50), "%t[ss1]", tooltip "Wie lange pro Schritt gewartet wird beim herunterfahren.", text variable: GV.p_Herunterfahren_Intervall
            OnMouseClick: write the text variable via VisuDialogs.Numpad
        Textfield (503,76 100x50), "s"
            OnMouseClick: write the text variable via Edit
    GroupBox (1041,752 768x181), "Inverter"
        Label (65,87 350x50), "IP-Adresse"
        Textfield (425,87 294x50), "%s", text variable: GV.p_Inverter_IP
            OnMouseClick: write the text variable via VisuDialogs.Numpad
    GroupBox (10,646 714x237), "Leistungsbegrenzung"
        Textfield (291,157 150x50), "%s", tooltip "Welche berechnete Drehzahl vom System verwendet wird.", text variable: GV.v_LeistungBegrenzung
            OnMouseClick: write the text variable via Default, min 0, max 3000
        Button (341,91 196x49), "Aktivieren"
            toggle GV.v_LeistungBegrenzung_ein
        Label (60,152 250x50), "Wert"
        Label (60,90 250x50), "Manuell"
    GroupBox (14,465 710x155), "Automatik"
        Button (149,67 380x49), "Aktivieren"
            toggle GV.p_Automatik
    Rectangle (0,0 1920x100)
    Button (944,19 300x60), "Parameter"
        OnMouseClick:  Assign=Parameter, Type=Assignment
    Button (324,19 300x60), "System"
        OnMouseClick:  Assign=System, Type=Assignment
    Button (634,19 300x60), "Elektrotechnik"
        OnMouseClick:  Assign=Elektrotechnik, Type=Assignment
    Button (14,19 300x60), "Übersicht"
        OnMouseClick:  Assign=Uebersicht, Type=Assignment
    Button (1254,19 300x60), "Log"
        OnMouseClick:  Assign=Logging, Type=Assignment
END_VISUALIZATION

// Visualisierung/Show
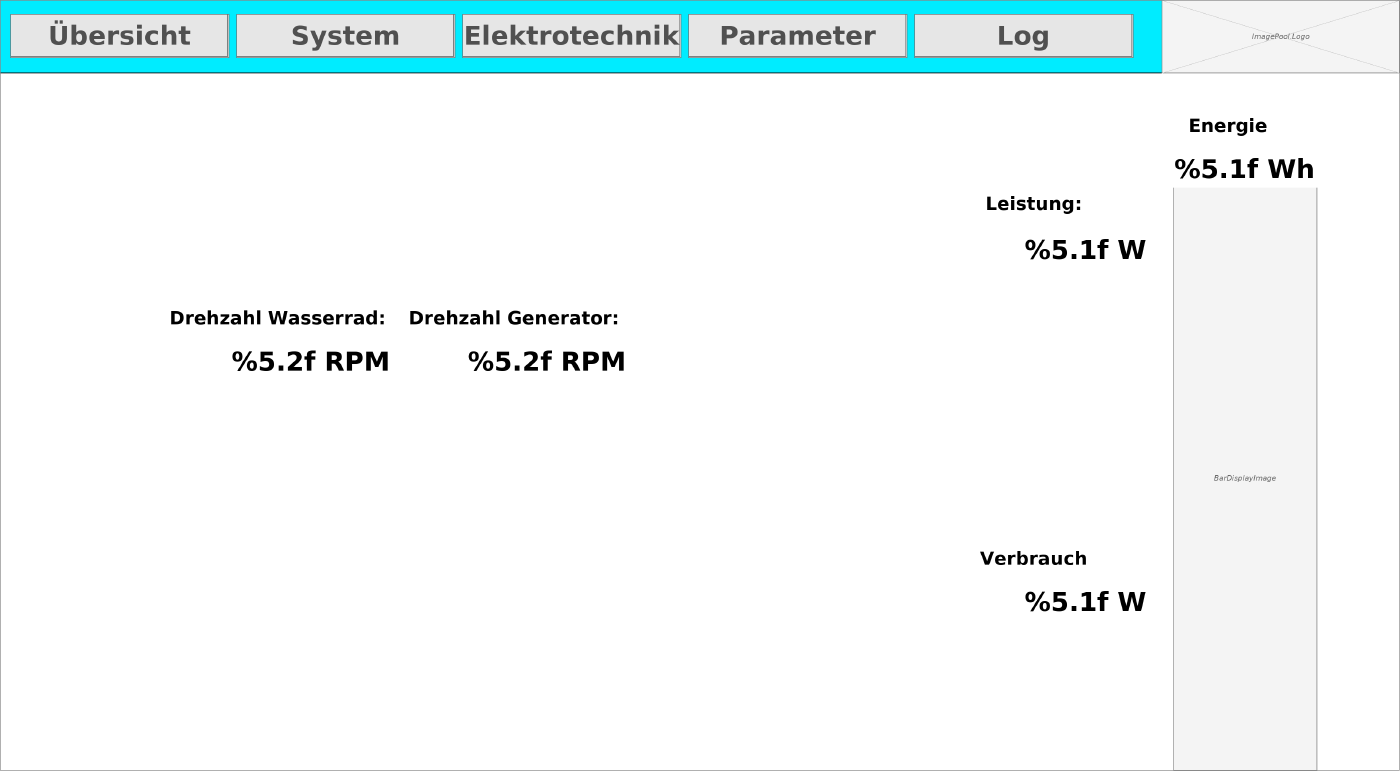
VISUALIZATION Show  // 1920x1058
    Rectangle (224,471 314x50), "%5.2f RPM", text variable: GV.sys_Drehzahl_Wasserrad
    Rectangle (1261,318 314x50), "%5.1f W", text variable: GV.r_LeistungAC
    Label (224,411 314x50), "Drehzahl Wasserrad:"
    Label (1261,254 314x50), "Leistung:"
    Rectangle (1555,891 150x30)
    BarDisplayImage (1609,254 197x804), value: GV.v_speicher, style: BarDisplayImage-Gray, scale format: %.1f, scale 0..300
    Label (1261,741 314x50), "Verbrauch"
    Rectangle (1261,801 314x50), "%5.1f W", text variable: GV.v_Kaffeemaschine
    Label (548,411 314x50), "Drehzahl Generator:"
    Rectangle (548,471 314x50), "%5.2f RPM", text variable: GV.sys_Drehzahl
    Label (1527,147 314x50), "Energie"
    Rectangle (1555,207 251x50), "%5.1f Wh", text variable: GV.v_speicher
    Rectangle (0,0 1920x100)
    Button (944,19 300x60), "Parameter"
        OnMouseClick:  Assign=Parameter, Type=Assignment
    Button (324,19 300x60), "System"
        OnMouseClick:  Assign=System, Type=Assignment
    Button (634,19 300x60), "Elektrotechnik"
        OnMouseClick:  Assign=Elektrotechnik, Type=Assignment
    Button (14,19 300x60), "Übersicht"
        OnMouseClick:  Assign=Uebersicht, Type=Assignment
    Button (1254,19 300x60), "Log"
        OnMouseClick:  Assign=Logging, Type=Assignment
    Image (1593,0 327x100), image: ImagePool.Logo
        OnMouseClick:  Assign=Info, Type=Assignment
END_VISUALIZATION

// Visualisierung/Logging
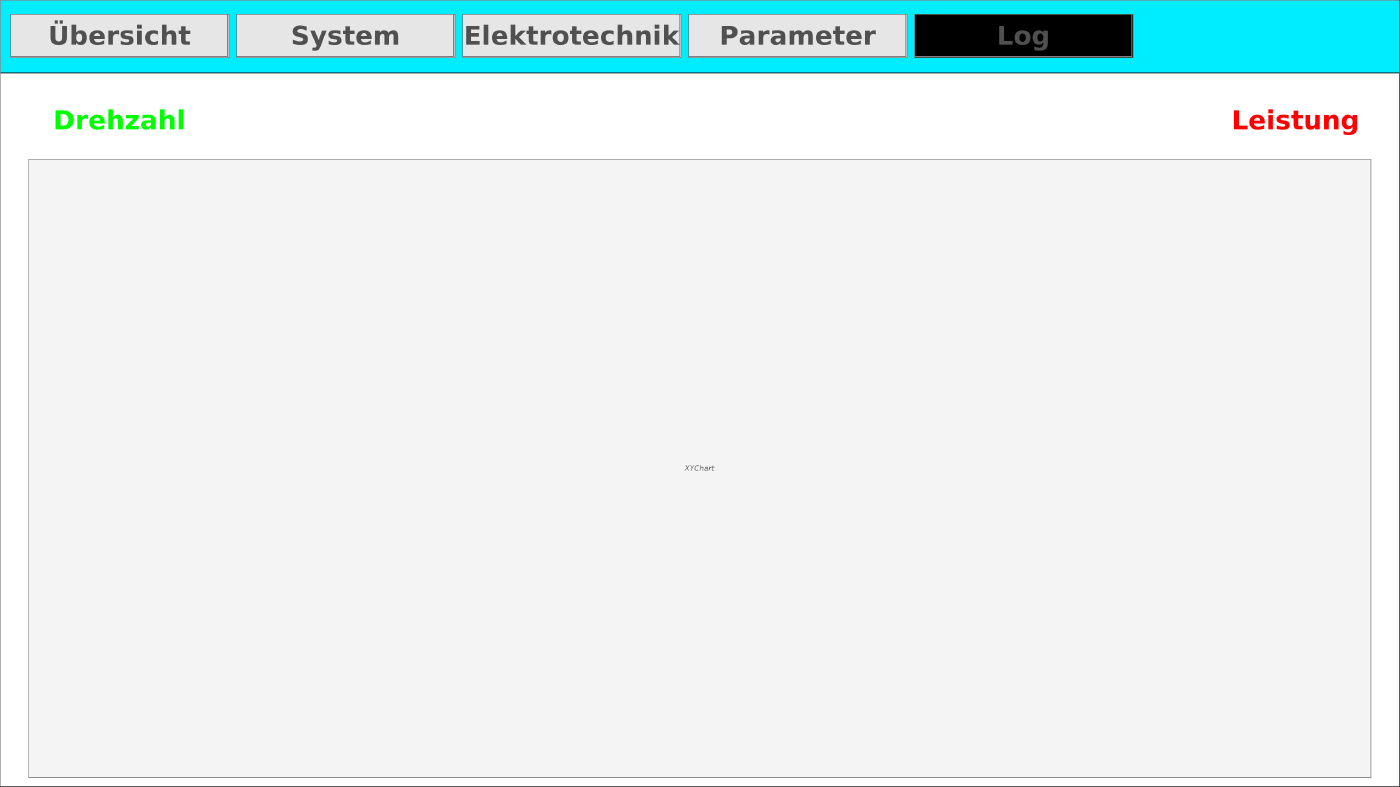
VISUALIZATION Logging  // 1920x1080
    Rectangle (0,0 1920x1080)
    Rectangle (0,0 1920x100)
    Button (944,19 300x60), "Parameter"
        OnMouseClick:  Assign=Parameter, Type=Assignment
    Button (324,19 300x60), "System"
        OnMouseClick:  Assign=System, Type=Assignment
    Button (634,19 300x60), "Elektrotechnik"
        OnMouseClick:  Assign=Elektrotechnik, Type=Assignment
    Button (14,19 300x60), "Übersicht"
        OnMouseClick:  Assign=Uebersicht, Type=Assignment
    XYChart (39,218 1841x849)
    Button (1254,19 300x60), "Log"
        OnMouseClick:  Assign=Logging, Type=Assignment
    Label (1667,150 220x30), "Leistung"
    Label (54,150 220x30), "Drehzahl"
END_VISUALIZATION

// Visualisierung/Info
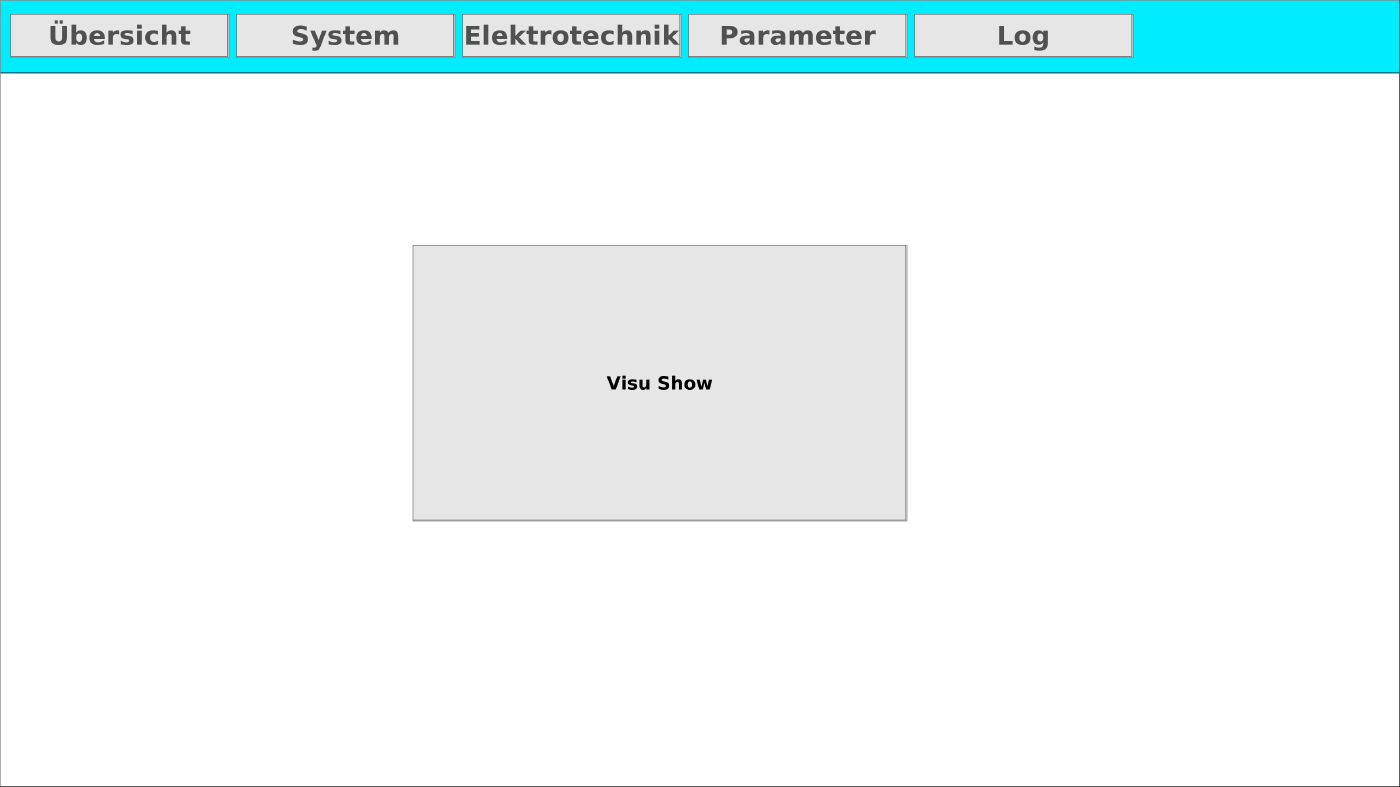
VISUALIZATION Info  // 1920x1080
    Rectangle (0,0 1920x1080)
    Rectangle (0,0 1920x100)
    Button (944,19 300x60), "Parameter"
        OnMouseClick:  Assign=Parameter, Type=Assignment
    Button (324,19 300x60), "System"
        OnMouseClick:  Assign=System, Type=Assignment
    Button (634,19 300x60), "Elektrotechnik"
        OnMouseClick:  Assign=Elektrotechnik, Type=Assignment
    Button (14,19 300x60), "Übersicht"
        OnMouseClick:  Assign=Uebersicht, Type=Assignment
    Button (1254,19 300x60), "Log"
        OnMouseClick:  Assign=Logging, Type=Assignment
    Button (566,336 678x379), "Visu Show"
        OnMouseClick:  Assign=Show, Type=Assignment
END_VISUALIZATION

